  MoveL 2674 to (229.6, 36.16, 50.44) mm, rotated rx -180 ry 0 rz 180 deg; joints [-27.455, 46.759, -73.474, 30.185, 113.51, 13.063]
  Call Extruder(589.48218)
  MoveL 2675 to (229.82, 36.23, 50.44) mm, rotated rx -180 ry 0 rz 180 deg; joints [-27.424, 46.781, -73.473, 30.147, 113.498, 13.038]
  MoveL 2676 to (229.82, 36.23, 50.44) mm, rotated rx -180 ry 0 rz 180 deg; joints [-27.424, 46.781, -73.473, 30.147, 113.498, 13.038]
  Call Extruder(589.60868)
  MoveL 2677 to (230.04, 36.29, 50.44) mm, rotated rx -180 ry 0 rz 180 deg; joints [-27.392, 46.804, -73.473, 30.108, 113.485, 13.012]
  MoveL 2678 to (230.04, 36.29, 50.44) mm, rotated rx -180 ry 0 rz 180 deg; joints [-27.392, 46.804, -73.473, 30.108, 113.485, 13.012]
  Call Extruder(589.73571)
  MoveL 2679 to (230.26, 36.36, 50.44) mm, rotated rx 180 ry 0 rz 180 deg; joints [-27.361, 46.826, -73.473, 30.07, 113.473, 12.986]
  MoveL 2680 to (230.26, 36.36, 50.44) mm, rotated rx 180 ry 0 rz 180 deg; joints [-27.361, 46.826, -73.473, 30.07, 113.473, 12.986]
  Call Extruder(589.86325)
  MoveL 2681 to (230.48, 36.42, 50.44) mm, rotated rx -180 ry 0 rz 180 deg; joints [-27.33, 46.848, -73.472, 30.032, 113.46, 12.961]
  MoveL 2682 to (230.48, 36.42, 50.44) mm, rotated rx -180 ry 0 rz 180 deg; joints [-27.33, 46.848, -73.472, 30.032, 113.46, 12.961]
  Call Extruder(589.99132)
  MoveL 2683 to (230.7, 36.49, 50.44) mm, rotated rx 180 ry 0 rz 180 deg; joints [-27.299, 46.87, -73.472, 29.994, 113.448, 12.935]
  MoveL 2684 to (230.7, 36.49, 50.44) mm, rotated rx 180 ry 0 rz 180 deg; joints [-27.299, 46.87, -73.472, 29.994, 113.448, 12.935]
  Call Extruder(590.10322)
  MoveL 2685 to (230.88, 36.55, 50.44) mm, rotated rx -180 ry 0 rz 180 deg; joints [-27.276, 46.89, -73.472, 29.966, 113.436, 12.915]
  MoveL 2686 to (230.88, 36.55, 50.44) mm, rotated rx -180 ry 0 rz 180 deg; joints [-27.276, 46.89, -73.472, 29.966, 113.436, 12.915]
  Call Extruder(590.21556)
  MoveL 2687 to (231.07, 36.61, 50.44) mm, rotated rx -180 ry 0 rz 180 deg; joints [-27.253, 46.909, -73.471, 29.937, 113.424, 12.894]
  MoveL 2688 to (231.07, 36.61, 50.44) mm, rotated rx -180 ry 0 rz 180 deg; joints [-27.253, 46.909, -73.471, 29.937, 113.424, 12.894]
  Call Extruder(590.32835)
  MoveL 2689 to (231.26, 36.67, 50.44) mm, rotated rx -180 ry 0 rz -180 deg; joints [-27.231, 46.929, -73.471, 29.909, 113.412, 12.874]
  MoveL 2690 to (231.26, 36.67, 50.44) mm, rotated rx -180 ry 0 rz -180 deg; joints [-27.231, 46.929, -73.471, 29.909, 113.412, 12.874]
  Call Extruder(590.44158)
  MoveL 2691 to (231.45, 36.73, 50.44) mm, rotated rx -180 ry 0 rz 180 deg; joints [-27.208, 46.948, -73.47, 29.88, 113.399, 12.854]
  MoveL 2692 to (231.45, 36.73, 50.44) mm, rotated rx -180 ry 0 rz 180 deg; joints [-27.208, 46.948, -73.47, 29.88, 113.399, 12.854]
  Call Extruder(590.55526)
  MoveL 2693 to (231.64, 36.79, 50.44) mm, rotated rx 180 ry 0 rz 180 deg; joints [-27.185, 46.967, -73.47, 29.852, 113.387, 12.834]
  MoveL 2694 to (231.64, 36.79, 50.44) mm, rotated rx 180 ry 0 rz 180 deg; joints [-27.185, 46.967, -73.47, 29.852, 113.387, 12.834]
  Call Extruder(590.73722)
  MoveL 2695 to (231.93, 36.91, 50.44) mm, rotated rx -180 ry 0 rz 180 deg; joints [-27.167, 46.999, -73.469, 29.826, 113.364, 12.809]
  MoveL 2696 to (231.93, 36.91, 50.44) mm, rotated rx -180 ry 0 rz 180 deg; joints [-27.167, 46.999, -73.469, 29.826, 113.364, 12.809]
  Call Extruder(590.91994)
  MoveL 2697 to (232.22, 37.04, 50.44) mm, rotated rx -180 ry 0 rz 180 deg; joints [-27.149, 47.03, -73.469, 29.8, 113.34, 12.784]
  MoveL 2698 to (232.22, 37.04, 50.44) mm, rotated rx -180 ry 0 rz 180 deg; joints [-27.149, 47.03, -73.469, 29.8, 113.34, 12.784]
  Call Extruder(591.09035)
  MoveL 2699 to (232.49, 37.15, 50.44) mm, rotated rx -180 ry 0 rz 180 deg; joints [-27.133, 47.059, -73.468, 29.777, 113.318, 12.761]
  MoveL 2700 to (232.49, 37.15, 50.44) mm, rotated rx -180 ry 0 rz 180 deg; joints [-27.133, 47.059, -73.468, 29.777, 113.318, 12.761]
  Call Extruder(591.24835)
  MoveL 2701 to (232.74, 37.26, 50.44) mm, rotated rx -180 ry 0 rz 180 deg; joints [-27.121, 47.085, -73.467, 29.758, 113.297, 12.741]
  MoveL 2702 to (232.74, 37.26, 50.44) mm, rotated rx -180 ry 0 rz 180 deg; joints [-27.121, 47.085, -73.467, 29.758, 113.297, 12.741]
  Call Extruder(591.40695)
  MoveL 2703 to (232.99, 37.36, 50.44) mm, rotated rx -180 ry 0 rz -180 deg; joints [-27.108, 47.112, -73.467, 29.738, 113.276, 12.721]
  MoveL 2704 to (232.99, 37.36, 50.44) mm, rotated rx -180 ry 0 rz -180 deg; joints [-27.108, 47.112, -73.467, 29.738, 113.276, 12.721]
  Call Extruder(591.61312)
  MoveL 2705 to (233.29, 37.54, 50.44) mm, rotated rx 180 ry 0 rz -180 deg; joints [-27.12, 47.147, -73.466, 29.743, 113.242, 12.707]
  MoveL 2706 to (233.29, 37.54, 50.44) mm, rotated rx 180 ry 0 rz -180 deg; joints [-27.12, 47.147, -73.466, 29.743, 113.242, 12.707]
  Call Extruder(591.82006)
  MoveL 2707 to (233.6, 37.71, 50.44) mm, rotated rx 180 ry 0 rz -180 deg; joints [-27.132, 47.181, -73.465, 29.749, 113.209, 12.693]
  MoveL 2708 to (233.6, 37.71, 50.44) mm, rotated rx 180 ry 0 rz -180 deg; joints [-27.132, 47.181, -73.465, 29.749, 113.209, 12.693]
  Call Extruder(592.02779)
  MoveL 2709 to (233.9, 37.89, 50.44) mm, rotated rx -180 ry 0 rz 180 deg; joints [-27.144, 47.216, -73.464, 29.754, 113.175, 12.678]
  MoveL 2710 to (233.9, 37.89, 50.44) mm, rotated rx -180 ry 0 rz 180 deg; joints [-27.144, 47.216, -73.464, 29.754, 113.175, 12.678]
  Call Extruder(592.23629)
  MoveL 2711 to (234.21, 38.07, 50.44) mm, rotated rx 180 ry 0 rz -180 deg; joints [-27.156, 47.251, -73.462, 29.759, 113.141, 12.664]
  MoveL 2712 to (234.21, 38.07, 50.44) mm, rotated rx 180 ry 0 rz -180 deg; joints [-27.156, 47.251, -73.462, 29.759, 113.141, 12.664]
  Call Extruder(592.41583)
  MoveL 2713 to (234.45, 38.24, 50.44) mm, rotated rx 180 ry 0 rz 180 deg; joints [-27.187, 47.28, -73.461, 29.785, 113.108, 12.661]
  MoveL 2714 to (234.45, 38.24, 50.44) mm, rotated rx 180 ry 0 rz 180 deg; joints [-27.187, 47.28, -73.461, 29.785, 113.108, 12.661]
  Call Extruder(592.74925)
  MoveL 2715 to (234.9, 38.57, 50.44) mm, rotated rx -180 ry 0 rz 180 deg; joints [-27.245, 47.334, -73.46, 29.835, 113.047, 12.655]
  MoveL 2716 to (234.9, 38.57, 50.44) mm, rotated rx -180 ry 0 rz 180 deg; joints [-27.245, 47.334, -73.46, 29.835, 113.047, 12.655]
  Call Extruder(593.08385)
  MoveL 2717 to (235.35, 38.9, 50.44) mm, rotated rx 180 ry 0 rz 180 deg; joints [-27.302, 47.388, -73.458, 29.884, 112.986, 12.648]
  Call Extruder(593.91180)
  MoveL 2718 to (236.39, 39.81, 50.44) mm, rotated rx -180 ry 0 rz 180 deg; joints [-27.525, 47.52, -73.452, 30.091, 112.819, 12.665]
  Call Extruder(594.73974)
  MoveL 2719 to (237.3, 40.85, 50.44) mm, rotated rx -180 ry 0 rz 180 deg; joints [-27.851, 47.646, -73.447, 30.408, 112.633, 12.727]
  Call Extruder(594.90704)
  MoveL 2720 to (237.47, 41.07, 50.44) mm, rotated rx -180 ry 0 rz 180 deg; joints [-27.932, 47.67, -73.445, 30.488, 112.593, 12.745]
  MoveL 2721 to (237.47, 41.07, 50.44) mm, rotated rx -180 ry 0 rz 180 deg; joints [-27.932, 47.67, -73.445, 30.488, 112.593, 12.745]
  Call Extruder(595.24045)
  MoveL 2722 to (237.8, 41.52, 50.44) mm, rotated rx 180 ry 0 rz -180 deg; joints [-28.091, 47.719, -73.443, 30.645, 112.514, 12.782]
  MoveL 2723 to (237.8, 41.52, 50.44) mm, rotated rx 180 ry 0 rz -180 deg; joints [-28.091, 47.719, -73.443, 30.645, 112.514, 12.782]
  Call Extruder(595.57268)
  MoveL 2724 to (238.12, 41.98, 50.44) mm, rotated rx -180 ry 0 rz 180 deg; joints [-28.249, 47.768, -73.44, 30.801, 112.434, 12.817]
  MoveL 2725 to (238.12, 41.98, 50.44) mm, rotated rx -180 ry 0 rz 180 deg; joints [-28.249, 47.768, -73.44, 30.801, 112.434, 12.817]
  Call Extruder(595.69039)
  MoveL 2726 to (238.22, 42.15, 50.44) mm, rotated rx -180 ry 0 rz 180 deg; joints [-28.315, 47.784, -73.439, 30.867, 112.405, 12.834]
  MoveL 2727 to (238.22, 42.15, 50.44) mm, rotated rx -180 ry 0 rz 180 deg; joints [-28.315, 47.784, -73.439, 30.867, 112.405, 12.834]
  Call Extruder(595.89811)
  MoveL 2728 to (238.4, 42.45, 50.44) mm, rotated rx 180 ry 0 rz 180 deg; joints [-28.434, 47.814, -73.438, 30.986, 112.352, 12.864]
  MoveL 2729 to (238.4, 42.45, 50.44) mm, rotated rx 180 ry 0 rz 180 deg; joints [-28.434, 47.814, -73.438, 30.986, 112.352, 12.864]
  Call Extruder(596.10507)
  MoveL 2730 to (238.57, 42.75, 50.44) mm, rotated rx 180 ry 0 rz 180 deg; joints [-28.552, 47.843, -73.436, 31.103, 112.3, 12.895]
  MoveL 2731 to (238.57, 42.75, 50.44) mm, rotated rx 180 ry 0 rz 180 deg; joints [-28.552, 47.843, -73.436, 31.103, 112.3, 12.895]
  Call Extruder(596.31124)
  MoveL 2732 to (238.75, 43.06, 50.44) mm, rotated rx -180 ry 0 rz 180 deg; joints [-28.669, 47.872, -73.435, 31.22, 112.247, 12.924]
  MoveL 2733 to (238.75, 43.06, 50.44) mm, rotated rx -180 ry 0 rz 180 deg; joints [-28.669, 47.872, -73.435, 31.22, 112.247, 12.924]
  Call Extruder(596.49292)
  MoveL 2734 to (238.89, 43.34, 50.44) mm, rotated rx -180 ry 0 rz 180 deg; joints [-28.78, 47.897, -73.433, 31.332, 112.2, 12.954]
  MoveL 2735 to (238.89, 43.34, 50.44) mm, rotated rx -180 ry 0 rz 180 deg; joints [-28.78, 47.897, -73.433, 31.332, 112.2, 12.954]
  Call Extruder(596.65093)
  MoveL 2736 to (239, 43.58, 50.44) mm, rotated rx 180 ry 0 rz 180 deg; joints [-28.886, 47.917, -73.432, 31.439, 112.157, 12.983]
  MoveL 2737 to (239, 43.58, 50.44) mm, rotated rx 180 ry 0 rz 180 deg; joints [-28.886, 47.917, -73.432, 31.439, 112.157, 12.983]
  Call Extruder(596.80833)
  MoveL 2738 to (239.11, 43.83, 50.44) mm, rotated rx -180 ry 0 rz 180 deg; joints [-28.991, 47.938, -73.431, 31.545, 112.115, 13.013]
  MoveL 2739 to (239.11, 43.83, 50.44) mm, rotated rx -180 ry 0 rz 180 deg; joints [-28.991, 47.938, -73.431, 31.545, 112.115, 13.013]
  Call Extruder(596.98254)
  MoveL 2740 to (239.22, 44.11, 50.44) mm, rotated rx -180 ry 0 rz 180 deg; joints [-29.11, 47.961, -73.429, 31.664, 112.067, 13.046]
  MoveL 2741 to (239.22, 44.11, 50.44) mm, rotated rx -180 ry 0 rz 180 deg; joints [-29.11, 47.961, -73.429, 31.664, 112.067, 13.046]
  Call Extruder(597.15607)
  MoveL 2742 to (239.33, 44.39, 50.44) mm, rotated rx -180 ry 0 rz 180 deg; joints [-29.228, 47.984, -73.428, 31.783, 112.02, 13.079]
  MoveL 2743 to (239.33, 44.39, 50.44) mm, rotated rx -180 ry 0 rz 180 deg; joints [-29.228, 47.984, -73.428, 31.783, 112.02, 13.079]
  Call Extruder(597.26356)
  MoveL 2744 to (239.41, 44.56, 50.44) mm, rotated rx -180 ry 0 rz 180 deg; joints [-29.301, 47.998, -73.427, 31.857, 111.991, 13.099]
  MoveL 2745 to (239.41, 44.56, 50.44) mm, rotated rx -180 ry 0 rz 180 deg; joints [-29.301, 47.998, -73.427, 31.857, 111.991, 13.099]
  Call Extruder(597.37703)
  MoveL 2746 to (239.47, 44.75, 50.44) mm, rotated rx -180 ry 0 rz -180 deg; joints [-29.385, 48.012, -73.426, 31.942, 111.959, 13.123]
  MoveL 2747 to (239.47, 44.75, 50.44) mm, rotated rx -180 ry 0 rz -180 deg; joints [-29.385, 48.012, -73.426, 31.942, 111.959, 13.123]
  Call Extruder(597.49005)
  MoveL 2748 to (239.53, 44.94, 50.44) mm, rotated rx -180 ry 0 rz 180 deg; joints [-29.47, 48.026, -73.425, 32.028, 111.927, 13.148]
  MoveL 2749 to (239.53, 44.94, 50.44) mm, rotated rx -180 ry 0 rz 180 deg; joints [-29.47, 48.026, -73.425, 32.028, 111.927, 13.148]
  Call Extruder(597.60263)
  MoveL 2750 to (239.59, 45.13, 50.44) mm, rotated rx 180 ry 0 rz -180 deg; joints [-29.553, 48.041, -73.424, 32.112, 111.895, 13.172]
  MoveL 2751 to (239.59, 45.13, 50.44) mm, rotated rx 180 ry 0 rz -180 deg; joints [-29.553, 48.041, -73.424, 32.112, 111.895, 13.172]
  Call Extruder(597.71477)
  MoveL 2752 to (239.65, 45.32, 50.44) mm, rotated rx 180 ry 0 rz 180 deg; joints [-29.637, 48.055, -73.423, 32.197, 111.863, 13.196]
  MoveL 2753 to (239.65, 45.32, 50.44) mm, rotated rx 180 ry 0 rz 180 deg; joints [-29.637, 48.055, -73.423, 32.197, 111.863, 13.196]
  Call Extruder(597.82645)
  MoveL 2754 to (239.71, 45.5, 50.44) mm, rotated rx -180 ry 0 rz 180 deg; joints [-29.72, 48.069, -73.422, 32.281, 111.831, 13.22]
  MoveL 2755 to (239.71, 45.5, 50.44) mm, rotated rx -180 ry 0 rz 180 deg; joints [-29.72, 48.069, -73.422, 32.281, 111.831, 13.22]
  Call Extruder(597.95753)
  MoveL 2756 to (239.78, 45.73, 50.44) mm, rotated rx 180 ry 0 rz 180 deg; joints [-29.821, 48.085, -73.421, 32.382, 111.794, 13.249]
  MoveL 2757 to (239.78, 45.73, 50.44) mm, rotated rx 180 ry 0 rz 180 deg; joints [-29.821, 48.085, -73.421, 32.382, 111.794, 13.249]
  Call Extruder(598.08804)
  MoveL 2758 to (239.85, 45.95, 50.44) mm, rotated rx 180 ry 0 rz 180 deg; joints [-29.921, 48.102, -73.42, 32.483, 111.756, 13.278]
  MoveL 2759 to (239.85, 45.95, 50.44) mm, rotated rx 180 ry 0 rz 180 deg; joints [-29.921, 48.102, -73.42, 32.483, 111.756, 13.278]
  Call Extruder(598.21798)
  MoveL 2760 to (239.92, 46.18, 50.44) mm, rotated rx -180 ry 0 rz 180 deg; joints [-30.02, 48.118, -73.419, 32.583, 111.718, 13.306]
  MoveL 2761 to (239.92, 46.18, 50.44) mm, rotated rx -180 ry 0 rz 180 deg; joints [-30.02, 48.118, -73.419, 32.583, 111.718, 13.306]
  Call Extruder(598.34736)
  MoveL 2762 to (239.98, 46.4, 50.44) mm, rotated rx 180 ry 0 rz -180 deg; joints [-30.119, 48.135, -73.418, 32.683, 111.681, 13.334]
  MoveL 2763 to (239.98, 46.4, 50.44) mm, rotated rx 180 ry 0 rz -180 deg; joints [-30.119, 48.135, -73.418, 32.683, 111.681, 13.334]
  Call Extruder(598.46931)
  MoveL 2764 to (240.04, 46.61, 50.44) mm, rotated rx -180 ry 0 rz 180 deg; joints [-30.216, 48.15, -73.417, 32.781, 111.645, 13.362]
  MoveL 2765 to (240.04, 46.61, 50.44) mm, rotated rx -180 ry 0 rz 180 deg; joints [-30.216, 48.15, -73.417, 32.781, 111.645, 13.362]
  Call Extruder(598.58414)
  MoveL 2766 to (240.08, 46.82, 50.44) mm, rotated rx -180 ry 0 rz 180 deg; joints [-30.311, 48.163, -73.416, 32.878, 111.61, 13.391]
  MoveL 2767 to (240.08, 46.82, 50.44) mm, rotated rx -180 ry 0 rz 180 deg; joints [-30.311, 48.163, -73.416, 32.878, 111.61, 13.391]
  Call Extruder(598.69851)
  MoveL 2768 to (240.13, 47.02, 50.44) mm, rotated rx -180 ry 0 rz 180 deg; joints [-30.406, 48.177, -73.415, 32.974, 111.576, 13.418]
  MoveL 2769 to (240.13, 47.02, 50.44) mm, rotated rx -180 ry 0 rz 180 deg; joints [-30.406, 48.177, -73.415, 32.974, 111.576, 13.418]
  Call Extruder(598.81243)
  MoveL 2770 to (240.17, 47.23, 50.44) mm, rotated rx -180 ry 0 rz 180 deg; joints [-30.5, 48.191, -73.414, 33.069, 111.542, 13.446]
  MoveL 2771 to (240.17, 47.23, 50.44) mm, rotated rx -180 ry 0 rz 180 deg; joints [-30.5, 48.191, -73.414, 33.069, 111.542, 13.446]
  Call Extruder(598.92591)
  MoveL 2772 to (240.22, 47.43, 50.44) mm, rotated rx -180 ry 0 rz 180 deg; joints [-30.595, 48.204, -73.413, 33.165, 111.508, 13.474]
  MoveL 2773 to (240.22, 47.43, 50.44) mm, rotated rx -180 ry 0 rz 180 deg; joints [-30.595, 48.204, -73.413, 33.165, 111.508, 13.474]
  Call Extruder(599.06319)
  MoveL 2774 to (240.27, 47.68, 50.44) mm, rotated rx -180 ry 0 rz 180 deg; joints [-30.711, 48.221, -73.412, 33.283, 111.466, 13.508]
  MoveL 2775 to (240.27, 47.68, 50.44) mm, rotated rx -180 ry 0 rz 180 deg; joints [-30.711, 48.221, -73.412, 33.283, 111.466, 13.508]
  Call Extruder(599.19986)
  MoveL 2776 to (240.32, 47.93, 50.44) mm, rotated rx -180 ry 0 rz 180 deg; joints [-30.827, 48.237, -73.411, 33.4, 111.424, 13.542]
  MoveL 2777 to (240.32, 47.93, 50.44) mm, rotated rx -180 ry 0 rz 180 deg; joints [-30.827, 48.237, -73.411, 33.4, 111.424, 13.542]
  Call Extruder(599.33592)
  MoveL 2778 to (240.37, 48.18, 50.44) mm, rotated rx -180 ry 0 rz 180 deg; joints [-30.942, 48.253, -73.409, 33.516, 111.383, 13.575]
  MoveL 2779 to (240.37, 48.18, 50.44) mm, rotated rx -180 ry 0 rz 180 deg; joints [-30.942, 48.253, -73.409, 33.516, 111.383, 13.575]
  Call Extruder(599.47137)
  MoveL 2780 to (240.42, 48.43, 50.44) mm, rotated rx -180 ry 0 rz 180 deg; joints [-31.057, 48.27, -73.408, 33.632, 111.341, 13.608]
  MoveL 2781 to (240.42, 48.43, 50.44) mm, rotated rx -180 ry 0 rz 180 deg; joints [-31.057, 48.27, -73.408, 33.632, 111.341, 13.608]
  Call Extruder(599.60622)
  MoveL 2782 to (240.47, 48.68, 50.44) mm, rotated rx 180 ry 0 rz 180 deg; joints [-31.171, 48.286, -73.407, 33.748, 111.299, 13.641]
  MoveL 2783 to (240.47, 48.68, 50.44) mm, rotated rx 180 ry 0 rz 180 deg; joints [-31.171, 48.286, -73.407, 33.748, 111.299, 13.641]
  Call Extruder(599.74045)
  MoveL 2784 to (240.52, 48.92, 50.44) mm, rotated rx -180 ry 0 rz 180 deg; joints [-31.285, 48.303, -73.406, 33.863, 111.258, 13.674]
  MoveL 2785 to (240.52, 48.92, 50.44) mm, rotated rx -180 ry 0 rz 180 deg; joints [-31.285, 48.303, -73.406, 33.863, 111.258, 13.674]
  Call Extruder(599.87407)
  MoveL 2786 to (240.57, 49.17, 50.44) mm, rotated rx -180 ry 0 rz 180 deg; joints [-31.398, 48.319, -73.405, 33.977, 111.216, 13.706]
  MoveL 2787 to (240.57, 49.17, 50.44) mm, rotated rx -180 ry 0 rz 180 deg; joints [-31.398, 48.319, -73.405, 33.977, 111.216, 13.706]
  Call Extruder(600.03618)
  MoveL 2788 to (240.61, 49.48, 50.44) mm, rotated rx 180 ry 0 rz 180 deg; joints [-31.541, 48.339, -73.403, 34.121, 111.165, 13.747]
  MoveL 2789 to (240.61, 49.48, 50.44) mm, rotated rx 180 ry 0 rz 180 deg; joints [-31.541, 48.339, -73.403, 34.121, 111.165, 13.747]
  Call Extruder(600.19756)
  MoveL 2790 to (240.66, 49.79, 50.44) mm, rotated rx -180 ry 0 rz 180 deg; joints [-31.684, 48.358, -73.402, 34.265, 111.114, 13.788]
  MoveL 2791 to (240.66, 49.79, 50.44) mm, rotated rx -180 ry 0 rz 180 deg; joints [-31.684, 48.358, -73.402, 34.265, 111.114, 13.788]
  Call Extruder(600.35821)
  MoveL 2792 to (240.71, 50.09, 50.44) mm, rotated rx -180 ry 0 rz 180 deg; joints [-31.825, 48.377, -73.4, 34.408, 111.063, 13.829]
  MoveL 2793 to (240.71, 50.09, 50.44) mm, rotated rx -180 ry 0 rz 180 deg; joints [-31.825, 48.377, -73.4, 34.408, 111.063, 13.829]
  Call Extruder(600.51814)
  MoveL 2794 to (240.76, 50.4, 50.44) mm, rotated rx -180 ry 0 rz 180 deg; joints [-31.966, 48.397, -73.398, 34.55, 111.012, 13.868]
  MoveL 2795 to (240.76, 50.4, 50.44) mm, rotated rx -180 ry 0 rz 180 deg; joints [-31.966, 48.397, -73.398, 34.55, 111.012, 13.868]
  Call Extruder(600.67734)
  MoveL 2796 to (240.81, 50.7, 50.44) mm, rotated rx -180 ry 0 rz 180 deg; joints [-32.106, 48.416, -73.397, 34.691, 110.961, 13.908]
  MoveL 2797 to (240.81, 50.7, 50.44) mm, rotated rx -180 ry 0 rz 180 deg; joints [-32.106, 48.416, -73.397, 34.691, 110.961, 13.908]
  Call Extruder(600.83580)
  MoveL 2798 to (240.86, 51.01, 50.44) mm, rotated rx 180 ry 0 rz 180 deg; joints [-32.246, 48.436, -73.395, 34.832, 110.91, 13.947]
  MoveL 2799 to (240.86, 51.01, 50.44) mm, rotated rx 180 ry 0 rz 180 deg; joints [-32.246, 48.436, -73.395, 34.832, 110.91, 13.947]
  Call Extruder(601.03468)
  MoveL 2800 to (240.9, 51.4, 50.44) mm, rotated rx -180 ry 0 rz 180 deg; joints [-32.427, 48.459, -73.393, 35.015, 110.845, 13.998]
  MoveL 2801 to (240.9, 51.4, 50.44) mm, rotated rx -180 ry 0 rz 180 deg; joints [-32.427, 48.459, -73.393, 35.015, 110.845, 13.998]
  Call Extruder(601.23269)
  MoveL 2802 to (240.95, 51.78, 50.44) mm, rotated rx -180 ry 0 rz 180 deg; joints [-32.608, 48.483, -73.391, 35.196, 110.78, 14.049]
  MoveL 2803 to (240.95, 51.78, 50.44) mm, rotated rx -180 ry 0 rz 180 deg; joints [-32.608, 48.483, -73.391, 35.196, 110.78, 14.049]
  Call Extruder(601.42983)
  MoveL 2804 to (240.99, 52.17, 50.44) mm, rotated rx -180 ry 0 rz 180 deg; joints [-32.787, 48.507, -73.389, 35.377, 110.716, 14.099]
  MoveL 2805 to (240.99, 52.17, 50.44) mm, rotated rx -180 ry 0 rz 180 deg; joints [-32.787, 48.507, -73.389, 35.377, 110.716, 14.099]
  Call Extruder(601.62610)
  MoveL 2806 to (241.04, 52.56, 50.44) mm, rotated rx -180 ry 0 rz -180 deg; joints [-32.966, 48.53, -73.387, 35.556, 110.651, 14.149]
  MoveL 2807 to (241.04, 52.56, 50.44) mm, rotated rx -180 ry 0 rz -180 deg; joints [-32.966, 48.53, -73.387, 35.556, 110.651, 14.149]
  Call Extruder(601.87181)
  MoveL 2808 to (241.09, 53.05, 50.44) mm, rotated rx 180 ry 0 rz 180 deg; joints [-33.193, 48.56, -73.385, 35.785, 110.57, 14.212]
  MoveL 2809 to (241.09, 53.05, 50.44) mm, rotated rx 180 ry 0 rz 180 deg; joints [-33.193, 48.56, -73.385, 35.785, 110.57, 14.212]
  Call Extruder(602.16658)
  MoveL 2810 to (241.13, 53.64, 50.44) mm, rotated rx 180 ry 0 rz 180 deg; joints [-33.469, 48.594, -73.382, 36.062, 110.471, 14.288]
  MoveL 2811 to (241.13, 53.64, 50.44) mm, rotated rx 180 ry 0 rz 180 deg; joints [-33.469, 48.594, -73.382, 36.062, 110.471, 14.288]
  Call Extruder(602.46002)
  MoveL 2812 to (241.18, 54.23, 50.44) mm, rotated rx -180 ry 0 rz 180 deg; joints [-33.742, 48.629, -73.379, 36.336, 110.373, 14.363]
  MoveL 2813 to (241.18, 54.23, 50.44) mm, rotated rx -180 ry 0 rz 180 deg; joints [-33.742, 48.629, -73.379, 36.336, 110.373, 14.363]
  Call Extruder(602.89337)
  MoveL 2814 to (241.23, 55.1, 50.44) mm, rotated rx -180 ry 0 rz 180 deg; joints [-34.152, 48.679, -73.374, 36.748, 110.227, 14.475]
  MoveL 2815 to (241.23, 55.1, 50.44) mm, rotated rx -180 ry 0 rz 180 deg; joints [-34.152, 48.679, -73.374, 36.748, 110.227, 14.475]
  Call Extruder(603.46554)
  MoveL 2816 to (241.27, 56.26, 50.44) mm, rotated rx -180 ry 0 rz 180 deg; joints [-34.696, 48.745, -73.368, 37.292, 110.033, 14.621]
  MoveL 2817 to (241.27, 56.26, 50.44) mm, rotated rx -180 ry 0 rz 180 deg; joints [-34.696, 48.745, -73.368, 37.292, 110.033, 14.621]
  Call Extruder(603.89324)
  MoveL 2818 to (241.29, 57.14, 50.44) mm, rotated rx 180 ry 0 rz 180 deg; joints [-35.104, 48.794, -73.363, 37.7, 109.887, 14.73]
  Call Extruder(645.88687)
  MoveL 2819 to (241.29, 142.86, 50.44) mm, rotated rx 180 ry 0 rz 180 deg; joints [-60.361, 54.458, -71.96, 61.513, 98.553, 15.326]
  MoveL 2820 to (241.29, 142.86, 50.44) mm, rotated rx 180 ry 0 rz 180 deg; joints [-60.361, 54.458, -71.96, 61.513, 98.553, 15.326]
  Call Extruder(646.60231)
  MoveL 2821 to (241.25, 144.32, 50.44) mm, rotated rx 180 ry 0 rz 180 deg; joints [-60.621, 54.556, -71.917, 61.749, 98.417, 15.239]
  MoveL 2822 to (241.25, 144.32, 50.44) mm, rotated rx 180 ry 0 rz 180 deg; joints [-60.621, 54.556, -71.917, 61.749, 98.417, 15.239]
  Call Extruder(647.17705)
  MoveL 2823 to (241.2, 145.48, 50.44) mm, rotated rx -180 ry 0 rz 180 deg; joints [-60.831, 54.634, -71.883, 61.939, 98.309, 15.169]
  MoveL 2824 to (241.2, 145.48, 50.44) mm, rotated rx -180 ry 0 rz 180 deg; joints [-60.831, 54.634, -71.883, 61.939, 98.309, 15.169]
  Call Extruder(647.47049)
  MoveL 2825 to (241.16, 146.07, 50.44) mm, rotated rx -180 ry 0 rz 180 deg; joints [-60.944, 54.673, -71.865, 62.042, 98.254, 15.135]
  MoveL 2826 to (241.16, 146.07, 50.44) mm, rotated rx -180 ry 0 rz 180 deg; joints [-60.944, 54.673, -71.865, 62.042, 98.254, 15.135]
  Call Extruder(647.76527)
  MoveL 2827 to (241.11, 146.66, 50.44) mm, rotated rx -180 ry 0 rz 180 deg; joints [-61.055, 54.711, -71.848, 62.144, 98.198, 15.1]
  MoveL 2828 to (241.11, 146.66, 50.44) mm, rotated rx -180 ry 0 rz 180 deg; joints [-61.055, 54.711, -71.848, 62.144, 98.198, 15.1]
  Call Extruder(648.06138)
  MoveL 2829 to (241.06, 147.25, 50.44) mm, rotated rx -180 ry 0 rz -180 deg; joints [-61.167, 54.75, -71.831, 62.245, 98.143, 15.066]
  MoveL 2830 to (241.06, 147.25, 50.44) mm, rotated rx -180 ry 0 rz -180 deg; joints [-61.167, 54.75, -71.831, 62.245, 98.143, 15.066]
  Call Extruder(648.25765)
  MoveL 2831 to (241.02, 147.63, 50.44) mm, rotated rx -180 ry 0 rz 180 deg; joints [-61.244, 54.775, -71.819, 62.316, 98.107, 15.044]
  MoveL 2832 to (241.02, 147.63, 50.44) mm, rotated rx -180 ry 0 rz 180 deg; joints [-61.244, 54.775, -71.819, 62.316, 98.107, 15.044]
  Call Extruder(648.45479)
  MoveL 2833 to (240.97, 148.02, 50.44) mm, rotated rx 180 ry 0 rz 180 deg; joints [-61.321, 54.799, -71.808, 62.386, 98.07, 15.023]
  MoveL 2834 to (240.97, 148.02, 50.44) mm, rotated rx 180 ry 0 rz 180 deg; joints [-61.321, 54.799, -71.808, 62.386, 98.07, 15.023]
  Call Extruder(648.65280)
  MoveL 2835 to (240.93, 148.41, 50.44) mm, rotated rx 180 ry 0 rz 180 deg; joints [-61.397, 54.824, -71.797, 62.457, 98.033, 15.001]
  MoveL 2836 to (240.93, 148.41, 50.44) mm, rotated rx 180 ry 0 rz 180 deg; joints [-61.397, 54.824, -71.797, 62.457, 98.033, 15.001]
  Call Extruder(648.85167)
  MoveL 2837 to (240.88, 148.8, 50.44) mm, rotated rx -180 ry 0 rz 180 deg; joints [-61.474, 54.849, -71.785, 62.527, 97.997, 14.979]
  MoveL 2838 to (240.88, 148.8, 50.44) mm, rotated rx -180 ry 0 rz 180 deg; joints [-61.474, 54.849, -71.785, 62.527, 97.997, 14.979]
  Call Extruder(649.03075)
  MoveL 2839 to (240.83, 149.14, 50.44) mm, rotated rx -180 ry 0 rz 180 deg; joints [-61.544, 54.871, -71.775, 62.591, 97.964, 14.96]
  MoveL 2840 to (240.83, 149.14, 50.44) mm, rotated rx -180 ry 0 rz 180 deg; joints [-61.544, 54.871, -71.775, 62.591, 97.964, 14.96]
  Call Extruder(649.18995)
  MoveL 2841 to (240.78, 149.45, 50.44) mm, rotated rx -180 ry 0 rz 180 deg; joints [-61.607, 54.89, -71.766, 62.649, 97.935, 14.943]
  MoveL 2842 to (240.78, 149.45, 50.44) mm, rotated rx -180 ry 0 rz 180 deg; joints [-61.607, 54.89, -71.766, 62.649, 97.935, 14.943]
  Call Extruder(649.34987)
  MoveL 2843 to (240.74, 149.76, 50.44) mm, rotated rx -180 ry 0 rz 180 deg; joints [-61.67, 54.909, -71.757, 62.708, 97.906, 14.927]
  MoveL 2844 to (240.74, 149.76, 50.44) mm, rotated rx -180 ry 0 rz 180 deg; joints [-61.67, 54.909, -71.757, 62.708, 97.906, 14.927]
  Call Extruder(649.51052)
  MoveL 2845 to (240.69, 150.06, 50.44) mm, rotated rx -180 ry 0 rz 180 deg; joints [-61.734, 54.928, -71.749, 62.766, 97.877, 14.91]
  MoveL 2846 to (240.69, 150.06, 50.44) mm, rotated rx -180 ry 0 rz 180 deg; joints [-61.734, 54.928, -71.749, 62.766, 97.877, 14.91]
  Call Extruder(649.67190)
  MoveL 2847 to (240.64, 150.37, 50.44) mm, rotated rx -180 ry 0 rz -180 deg; joints [-61.796, 54.947, -71.74, 62.824, 97.848, 14.893]
  MoveL 2848 to (240.64, 150.37, 50.44) mm, rotated rx -180 ry 0 rz -180 deg; joints [-61.796, 54.947, -71.74, 62.824, 97.848, 14.893]
  Call Extruder(649.83401)
  MoveL 2849 to (240.59, 150.67, 50.44) mm, rotated rx -180 ry 0 rz 180 deg; joints [-61.859, 54.966, -71.731, 62.882, 97.819, 14.876]
  MoveL 2850 to (240.59, 150.67, 50.44) mm, rotated rx -180 ry 0 rz 180 deg; joints [-61.859, 54.966, -71.731, 62.882, 97.819, 14.876]
  Call Extruder(649.98221)
  MoveL 2851 to (240.54, 150.95, 50.44) mm, rotated rx 180 ry 0 rz 180 deg; joints [-61.918, 54.983, -71.723, 62.936, 97.792, 14.862]
  MoveL 2852 to (240.54, 150.95, 50.44) mm, rotated rx 180 ry 0 rz 180 deg; joints [-61.918, 54.983, -71.723, 62.936, 97.792, 14.862]
  Call Extruder(650.11644)
  MoveL 2853 to (240.49, 151.2, 50.44) mm, rotated rx -180 ry 0 rz 180 deg; joints [-61.971, 54.998, -71.715, 62.985, 97.768, 14.848]
  MoveL 2854 to (240.49, 151.2, 50.44) mm, rotated rx -180 ry 0 rz 180 deg; joints [-61.971, 54.998, -71.715, 62.985, 97.768, 14.848]
  Call Extruder(650.25129)
  MoveL 2855 to (240.44, 151.45, 50.44) mm, rotated rx -180 ry 0 rz 180 deg; joints [-62.025, 55.013, -71.708, 63.035, 97.745, 14.836]
  MoveL 2856 to (240.44, 151.45, 50.44) mm, rotated rx -180 ry 0 rz 180 deg; joints [-62.025, 55.013, -71.708, 63.035, 97.745, 14.836]
  Call Extruder(650.38674)
  MoveL 2857 to (240.39, 151.7, 50.44) mm, rotated rx 180 ry 0 rz 180 deg; joints [-62.079, 55.028, -71.701, 63.084, 97.721, 14.822]
  MoveL 2858 to (240.39, 151.7, 50.44) mm, rotated rx 180 ry 0 rz 180 deg; joints [-62.079, 55.028, -71.701, 63.084, 97.721, 14.822]
  Call Extruder(650.52280)
  MoveL 2859 to (240.34, 151.95, 50.44) mm, rotated rx -180 ry 0 rz -180 deg; joints [-62.132, 55.044, -71.694, 63.134, 97.697, 14.809]
  MoveL 2860 to (240.34, 151.95, 50.44) mm, rotated rx -180 ry 0 rz -180 deg; joints [-62.132, 55.044, -71.694, 63.134, 97.697, 14.809]
  Call Extruder(650.65947)
  MoveL 2861 to (240.29, 152.2, 50.44) mm, rotated rx -180 ry 0 rz -180 deg; joints [-62.186, 55.059, -71.686, 63.183, 97.673, 14.796]
  MoveL 2862 to (240.29, 152.2, 50.44) mm, rotated rx -180 ry 0 rz -180 deg; joints [-62.186, 55.059, -71.686, 63.183, 97.673, 14.796]
  Call Extruder(650.79675)
  MoveL 2863 to (240.24, 152.44, 50.44) mm, rotated rx -180 ry 0 rz 180 deg; joints [-62.239, 55.074, -71.679, 63.233, 97.649, 14.783]
  MoveL 2864 to (240.24, 152.44, 50.44) mm, rotated rx -180 ry 0 rz 180 deg; joints [-62.239, 55.074, -71.679, 63.233, 97.649, 14.783]
  Call Extruder(650.92242)
  MoveL 2865 to (240.2, 152.67, 50.44) mm, rotated rx -180 ry 0 rz 180 deg; joints [-62.288, 55.088, -71.673, 63.278, 97.628, 14.771]
  MoveL 2866 to (240.2, 152.67, 50.44) mm, rotated rx -180 ry 0 rz 180 deg; joints [-62.288, 55.088, -71.673, 63.278, 97.628, 14.771]
  Call Extruder(651.03634)
  MoveL 2867 to (240.15, 152.88, 50.44) mm, rotated rx -180 ry 0 rz 180 deg; joints [-62.333, 55.1, -71.667, 63.319, 97.608, 14.76]
  MoveL 2868 to (240.15, 152.88, 50.44) mm, rotated rx -180 ry 0 rz 180 deg; joints [-62.333, 55.1, -71.667, 63.319, 97.608, 14.76]
  Call Extruder(651.15072)
  MoveL 2869 to (240.11, 153.08, 50.44) mm, rotated rx -180 ry 0 rz 180 deg; joints [-62.377, 55.112, -71.661, 63.36, 97.589, 14.749]
  MoveL 2870 to (240.11, 153.08, 50.44) mm, rotated rx -180 ry 0 rz 180 deg; joints [-62.377, 55.112, -71.661, 63.36, 97.589, 14.749]
  Call Extruder(651.26555)
  MoveL 2871 to (240.06, 153.28, 50.44) mm, rotated rx -180 ry 0 rz 180 deg; joints [-62.421, 55.124, -71.655, 63.402, 97.569, 14.739]
  MoveL 2872 to (240.06, 153.28, 50.44) mm, rotated rx -180 ry 0 rz 180 deg; joints [-62.421, 55.124, -71.655, 63.402, 97.569, 14.739]
  Call Extruder(651.38083)
  MoveL 2873 to (240.02, 153.49, 50.44) mm, rotated rx -180 ry 0 rz 180 deg; joints [-62.466, 55.137, -71.649, 63.443, 97.55, 14.728]
  MoveL 2874 to (240.02, 153.49, 50.44) mm, rotated rx -180 ry 0 rz 180 deg; joints [-62.466, 55.137, -71.649, 63.443, 97.55, 14.728]
  Call Extruder(651.51021)
  MoveL 2875 to (239.95, 153.71, 50.44) mm, rotated rx 180 ry 0 rz 180 deg; joints [-62.52, 55.15, -71.642, 63.493, 97.527, 14.718]
  MoveL 2876 to (239.95, 153.71, 50.44) mm, rotated rx 180 ry 0 rz 180 deg; joints [-62.52, 55.15, -71.642, 63.493, 97.527, 14.718]
  Call Extruder(651.64015)
  MoveL 2877 to (239.88, 153.94, 50.44) mm, rotated rx -180 ry 0 rz -180 deg; joints [-62.574, 55.162, -71.636, 63.544, 97.505, 14.707]
  MoveL 2878 to (239.88, 153.94, 50.44) mm, rotated rx -180 ry 0 rz -180 deg; joints [-62.574, 55.162, -71.636, 63.544, 97.505, 14.707]
  Call Extruder(651.77066)
  MoveL 2879 to (239.81, 154.16, 50.44) mm, rotated rx -180 ry 0 rz 180 deg; joints [-62.627, 55.175, -71.63, 63.594, 97.483, 14.697]
  MoveL 2880 to (239.81, 154.16, 50.44) mm, rotated rx -180 ry 0 rz 180 deg; joints [-62.627, 55.175, -71.63, 63.594, 97.483, 14.697]
  Call Extruder(651.90174)
  MoveL 2881 to (239.75, 154.38, 50.44) mm, rotated rx -180 ry 0 rz 180 deg; joints [-62.681, 55.188, -71.624, 63.644, 97.461, 14.686]
  MoveL 2882 to (239.75, 154.38, 50.44) mm, rotated rx -180 ry 0 rz 180 deg; joints [-62.681, 55.188, -71.624, 63.644, 97.461, 14.686]
  Call Extruder(652.02338)
  MoveL 2883 to (239.68, 154.59, 50.44) mm, rotated rx 180 ry 0 rz 180 deg; joints [-62.731, 55.2, -71.618, 63.691, 97.441, 14.677]
  MoveL 2884 to (239.68, 154.59, 50.44) mm, rotated rx 180 ry 0 rz 180 deg; joints [-62.731, 55.2, -71.618, 63.691, 97.441, 14.677]
  Call Extruder(652.13550)
  MoveL 2885 to (239.62, 154.78, 50.44) mm, rotated rx 180 ry 0 rz 180 deg; joints [-62.778, 55.21, -71.613, 63.734, 97.422, 14.668]
  MoveL 2886 to (239.62, 154.78, 50.44) mm, rotated rx 180 ry 0 rz 180 deg; joints [-62.778, 55.21, -71.613, 63.734, 97.422, 14.668]
  Call Extruder(652.24807)
  MoveL 2887 to (239.56, 154.97, 50.44) mm, rotated rx -180 ry 0 rz 180 deg; joints [-62.824, 55.221, -71.607, 63.777, 97.403, 14.66]
  MoveL 2888 to (239.56, 154.97, 50.44) mm, rotated rx -180 ry 0 rz 180 deg; joints [-62.824, 55.221, -71.607, 63.777, 97.403, 14.66]
  Call Extruder(652.36108)
  MoveL 2889 to (239.5, 155.15, 50.44) mm, rotated rx -180 ry 0 rz 180 deg; joints [-62.87, 55.232, -71.602, 63.821, 97.384, 14.651]
  MoveL 2890 to (239.5, 155.15, 50.44) mm, rotated rx -180 ry 0 rz 180 deg; joints [-62.87, 55.232, -71.602, 63.821, 97.384, 14.651]
  Call Extruder(652.47454)
  MoveL 2891 to (239.44, 155.34, 50.44) mm, rotated rx 180 ry 0 rz 180 deg; joints [-62.916, 55.242, -71.597, 63.864, 97.366, 14.643]
  MoveL 2892 to (239.44, 155.34, 50.44) mm, rotated rx 180 ry 0 rz 180 deg; joints [-62.916, 55.242, -71.597, 63.864, 97.366, 14.643]
  Call Extruder(652.62218)
  MoveL 2893 to (239.35, 155.58, 50.44) mm, rotated rx -180 ry 0 rz 180 deg; joints [-62.979, 55.255, -71.59, 63.923, 97.341, 14.633]
  MoveL 2894 to (239.35, 155.58, 50.44) mm, rotated rx -180 ry 0 rz 180 deg; joints [-62.979, 55.255, -71.59, 63.923, 97.341, 14.633]
  Call Extruder(652.80452)
  MoveL 2895 to (239.22, 155.87, 50.44) mm, rotated rx -180 ry 0 rz 180 deg; joints [-63.058, 55.271, -71.582, 63.997, 97.311, 14.621]
  MoveL 2896 to (239.22, 155.87, 50.44) mm, rotated rx -180 ry 0 rz 180 deg; joints [-63.058, 55.271, -71.582, 63.997, 97.311, 14.621]
  Call Extruder(652.98761)
  MoveL 2897 to (239.1, 156.17, 50.44) mm, rotated rx 180 ry 0 rz 180 deg; joints [-63.136, 55.287, -71.575, 64.07, 97.281, 14.609]
  MoveL 2898 to (239.1, 156.17, 50.44) mm, rotated rx 180 ry 0 rz 180 deg; joints [-63.136, 55.287, -71.575, 64.07, 97.281, 14.609]
  Call Extruder(653.14533)
  MoveL 2899 to (239, 156.42, 50.44) mm, rotated rx 180 ry 0 rz 180 deg; joints [-63.204, 55.3, -71.568, 64.135, 97.255, 14.6]
  MoveL 2900 to (239, 156.42, 50.44) mm, rotated rx 180 ry 0 rz 180 deg; joints [-63.204, 55.3, -71.568, 64.135, 97.255, 14.6]
  Call Extruder(653.30365)
  MoveL 2901 to (238.89, 156.66, 50.44) mm, rotated rx 180 ry 0 rz 180 deg; joints [-63.272, 55.313, -71.561, 64.198, 97.229, 14.59]
  MoveL 2902 to (238.89, 156.66, 50.44) mm, rotated rx 180 ry 0 rz 180 deg; joints [-63.272, 55.313, -71.561, 64.198, 97.229, 14.59]
  Call Extruder(653.48569)
  MoveL 2903 to (238.75, 156.94, 50.44) mm, rotated rx -180 ry 0 rz -180 deg; joints [-63.354, 55.327, -71.554, 64.276, 97.2, 14.581]
  MoveL 2904 to (238.75, 156.94, 50.44) mm, rotated rx -180 ry 0 rz -180 deg; joints [-63.354, 55.327, -71.554, 64.276, 97.2, 14.581]
  Call Extruder(653.69224)
  MoveL 2905 to (238.57, 157.25, 50.44) mm, rotated rx 180 ry 0 rz 180 deg; joints [-63.449, 55.342, -71.547, 64.367, 97.166, 14.573]
  MoveL 2906 to (238.57, 157.25, 50.44) mm, rotated rx 180 ry 0 rz 180 deg; joints [-63.449, 55.342, -71.547, 64.367, 97.166, 14.573]
  Call Extruder(653.89957)
  MoveL 2907 to (238.4, 157.55, 50.44) mm, rotated rx -180 ry 0 rz 180 deg; joints [-63.544, 55.357, -71.539, 64.457, 97.132, 14.564]
  MoveL 2908 to (238.4, 157.55, 50.44) mm, rotated rx -180 ry 0 rz 180 deg; joints [-63.544, 55.357, -71.539, 64.457, 97.132, 14.564]
  Call Extruder(654.10768)
  MoveL 2909 to (238.22, 157.85, 50.44) mm, rotated rx -180 ry 0 rz 180 deg; joints [-63.64, 55.371, -71.532, 64.547, 97.099, 14.556]
  MoveL 2910 to (238.22, 157.85, 50.44) mm, rotated rx -180 ry 0 rz 180 deg; joints [-63.64, 55.371, -71.532, 64.547, 97.099, 14.556]
  Call Extruder(654.22535)
  MoveL 2911 to (238.12, 158.02, 50.44) mm, rotated rx -180 ry 0 rz 180 deg; joints [-63.693, 55.38, -71.528, 64.598, 97.08, 14.551]
  MoveL 2912 to (238.12, 158.02, 50.44) mm, rotated rx -180 ry 0 rz 180 deg; joints [-63.693, 55.38, -71.528, 64.598, 97.08, 14.551]
  Call Extruder(654.55818)
  MoveL 2913 to (237.79, 158.48, 50.44) mm, rotated rx 180 ry 0 rz 180 deg; joints [-63.854, 55.399, -71.518, 64.752, 97.027, 14.543]
  MoveL 2914 to (237.79, 158.48, 50.44) mm, rotated rx 180 ry 0 rz 180 deg; joints [-63.854, 55.399, -71.518, 64.752, 97.027, 14.543]
  Call Extruder(654.89221)
  MoveL 2915 to (237.47, 158.93, 50.44) mm, rotated rx -180 ry 0 rz -180 deg; joints [-64.014, 55.419, -71.508, 64.904, 96.974, 14.535]
  MoveL 2916 to (237.47, 158.93, 50.44) mm, rotated rx -180 ry 0 rz -180 deg; joints [-64.014, 55.419, -71.508, 64.904, 96.974, 14.535]
  Call Extruder(655.05980)
  MoveL 2917 to (237.3, 159.15, 50.44) mm, rotated rx -180 ry 0 rz 180 deg; joints [-64.094, 55.429, -71.503, 64.98, 96.948, 14.53]
  Call Extruder(655.88912)
  MoveL 2918 to (236.39, 160.19, 50.44) mm, rotated rx 180 ry 0 rz 180 deg; joints [-64.505, 55.47, -71.482, 65.375, 96.819, 14.522]
  Call Extruder(656.52018)
  MoveL 2919 to (235.6, 160.89, 50.44) mm, rotated rx -180 ry 0 rz 180 deg; joints [-64.83, 55.492, -71.47, 65.688, 96.723, 14.529]
  MoveL 2920 to (235.6, 160.89, 50.44) mm, rotated rx -180 ry 0 rz 180 deg; joints [-64.83, 55.492, -71.47, 65.688, 96.723, 14.529]
  Call Extruder(656.71780)
  MoveL 2921 to (235.35, 161.1, 50.44) mm, rotated rx -180 ry 0 rz 180 deg; joints [-64.933, 55.498, -71.467, 65.787, 96.693, 14.531]
  Call Extruder(657.05182)
  MoveL 2922 to (234.9, 161.43, 50.44) mm, rotated rx -180 ry 0 rz 180 deg; joints [-65.109, 55.506, -71.463, 65.958, 96.644, 14.54]
  MoveL 2923 to (234.9, 161.43, 50.44) mm, rotated rx -180 ry 0 rz 180 deg; joints [-65.109, 55.506, -71.463, 65.958, 96.644, 14.54]
  Call Extruder(657.38465)
  MoveL 2924 to (234.45, 161.76, 50.44) mm, rotated rx -180 ry 0 rz 180 deg; joints [-65.285, 55.515, -71.458, 66.128, 96.595, 14.548]
  MoveL 2925 to (234.45, 161.76, 50.44) mm, rotated rx -180 ry 0 rz 180 deg; joints [-65.285, 55.515, -71.458, 66.128, 96.595, 14.548]
  Call Extruder(657.56385)
  MoveL 2926 to (234.21, 161.94, 50.44) mm, rotated rx 180 ry 0 rz -180 deg; joints [-65.381, 55.519, -71.456, 66.22, 96.568, 14.553]
  MoveL 2927 to (234.21, 161.94, 50.44) mm, rotated rx 180 ry 0 rz -180 deg; joints [-65.381, 55.519, -71.456, 66.22, 96.568, 14.553]
  Call Extruder(657.77197)
  MoveL 2928 to (233.9, 162.11, 50.44) mm, rotated rx 180 ry 0 rz 180 deg; joints [-65.493, 55.521, -71.455, 66.329, 96.539, 14.562]
  MoveL 2929 to (233.9, 162.11, 50.44) mm, rotated rx 180 ry 0 rz 180 deg; joints [-65.493, 55.521, -71.455, 66.329, 96.539, 14.562]
  Call Extruder(657.97930)
  MoveL 2930 to (233.6, 162.29, 50.44) mm, rotated rx 180 ry 0 rz -180 deg; joints [-65.605, 55.524, -71.453, 66.438, 96.509, 14.571]
  MoveL 2931 to (233.6, 162.29, 50.44) mm, rotated rx 180 ry 0 rz -180 deg; joints [-65.605, 55.524, -71.453, 66.438, 96.509, 14.571]
  Call Extruder(658.18586)
  MoveL 2932 to (233.29, 162.46, 50.44) mm, rotated rx 180 ry 0 rz 180 deg; joints [-65.718, 55.527, -71.452, 66.547, 96.479, 14.579]
  MoveL 2933 to (233.29, 162.46, 50.44) mm, rotated rx 180 ry 0 rz 180 deg; joints [-65.718, 55.527, -71.452, 66.547, 96.479, 14.579]
  Call Extruder(658.39164)
  MoveL 2934 to (232.99, 162.64, 50.44) mm, rotated rx 180 ry 0 rz 180 deg; joints [-65.83, 55.529, -71.451, 66.656, 96.449, 14.588]
  MoveL 2935 to (232.99, 162.64, 50.44) mm, rotated rx 180 ry 0 rz 180 deg; joints [-65.83, 55.529, -71.451, 66.656, 96.449, 14.588]
  Call Extruder(658.54991)
  MoveL 2936 to (232.74, 162.74, 50.44) mm, rotated rx -180 ry 0 rz 180 deg; joints [-65.917, 55.529, -71.451, 66.741, 96.427, 14.598]
  MoveL 2937 to (232.74, 162.74, 50.44) mm, rotated rx -180 ry 0 rz 180 deg; joints [-65.917, 55.529, -71.451, 66.741, 96.427, 14.598]
  Call Extruder(658.70759)
  MoveL 2938 to (232.49, 162.85, 50.44) mm, rotated rx 180 ry 0 rz -180 deg; joints [-66.004, 55.529, -71.451, 66.826, 96.405, 14.608]
  MoveL 2939 to (232.49, 162.85, 50.44) mm, rotated rx 180 ry 0 rz -180 deg; joints [-66.004, 55.529, -71.451, 66.826, 96.405, 14.608]
  Call Extruder(658.87768)
  MoveL 2940 to (232.22, 162.96, 50.44) mm, rotated rx 180 ry 0 rz 180 deg; joints [-66.099, 55.528, -71.451, 66.918, 96.382, 14.619]
  MoveL 2941 to (232.22, 162.96, 50.44) mm, rotated rx 180 ry 0 rz 180 deg; joints [-66.099, 55.528, -71.451, 66.918, 96.382, 14.619]
  Call Extruder(659.06004)
  MoveL 2942 to (231.93, 163.09, 50.44) mm, rotated rx -180 ry 0 rz 180 deg; joints [-66.2, 55.528, -71.451, 67.017, 96.357, 14.63]
  MoveL 2943 to (231.93, 163.09, 50.44) mm, rotated rx -180 ry 0 rz 180 deg; joints [-66.2, 55.528, -71.451, 67.017, 96.357, 14.63]
  Call Extruder(659.24164)
  MoveL 2944 to (231.64, 163.21, 50.44) mm, rotated rx 180 ry 0 rz 180 deg; joints [-66.302, 55.527, -71.452, 67.116, 96.331, 14.642]
  MoveL 2945 to (231.64, 163.21, 50.44) mm, rotated rx 180 ry 0 rz 180 deg; joints [-66.302, 55.527, -71.452, 67.116, 96.331, 14.642]
  Call Extruder(659.35509)
  MoveL 2946 to (231.45, 163.27, 50.44) mm, rotated rx 180 ry 0 rz -180 deg; joints [-66.365, 55.526, -71.452, 67.178, 96.316, 14.651]
  MoveL 2947 to (231.45, 163.27, 50.44) mm, rotated rx 180 ry 0 rz -180 deg; joints [-66.365, 55.526, -71.452, 67.178, 96.316, 14.651]
  Call Extruder(659.46809)
  MoveL 2948 to (231.26, 163.33, 50.44) mm, rotated rx 180 ry 0 rz 180 deg; joints [-66.428, 55.524, -71.453, 67.24, 96.301, 14.66]
  MoveL 2949 to (231.26, 163.33, 50.44) mm, rotated rx 180 ry 0 rz 180 deg; joints [-66.428, 55.524, -71.453, 67.24, 96.301, 14.66]
  Call Extruder(659.58064)
  MoveL 2950 to (231.07, 163.39, 50.44) mm, rotated rx -180 ry 0 rz 180 deg; joints [-66.492, 55.523, -71.454, 67.302, 96.286, 14.668]
  MoveL 2951 to (231.07, 163.39, 50.44) mm, rotated rx -180 ry 0 rz 180 deg; joints [-66.492, 55.523, -71.454, 67.302, 96.286, 14.668]
  Call Extruder(659.69275)
  MoveL 2952 to (230.88, 163.45, 50.44) mm, rotated rx -180 ry 0 rz -180 deg; joints [-66.555, 55.521, -71.455, 67.364, 96.27, 14.677]
  MoveL 2953 to (230.88, 163.45, 50.44) mm, rotated rx -180 ry 0 rz -180 deg; joints [-66.555, 55.521, -71.455, 67.364, 96.27, 14.677]
  Call Extruder(659.80442)
  MoveL 2954 to (230.69, 163.51, 50.44) mm, rotated rx -180 ry 0 rz -180 deg; joints [-66.619, 55.52, -71.455, 67.426, 96.255, 14.686]
  MoveL 2955 to (230.69, 163.51, 50.44) mm, rotated rx -180 ry 0 rz -180 deg; joints [-66.619, 55.52, -71.455, 67.426, 96.255, 14.686]
  Call Extruder(659.93552)
  MoveL 2956 to (230.47, 163.58, 50.44) mm, rotated rx -180 ry 0 rz 180 deg; joints [-66.694, 55.518, -71.457, 67.499, 96.237, 14.697]
  MoveL 2957 to (230.47, 163.58, 50.44) mm, rotated rx -180 ry 0 rz 180 deg; joints [-66.694, 55.518, -71.457, 67.499, 96.237, 14.697]
  Call Extruder(660.06605)
  MoveL 2958 to (230.25, 163.65, 50.44) mm, rotated rx -180 ry 0 rz -180 deg; joints [-66.768, 55.516, -71.458, 67.572, 96.22, 14.707]
  MoveL 2959 to (230.25, 163.65, 50.44) mm, rotated rx -180 ry 0 rz -180 deg; joints [-66.768, 55.516, -71.458, 67.572, 96.22, 14.707]
  Call Extruder(660.19601)
  MoveL 2960 to (230.02, 163.72, 50.44) mm, rotated rx -180 ry 0 rz 180 deg; joints [-66.843, 55.514, -71.459, 67.645, 96.202, 14.718]
  MoveL 2961 to (230.02, 163.72, 50.44) mm, rotated rx -180 ry 0 rz 180 deg; joints [-66.843, 55.514, -71.459, 67.645, 96.202, 14.718]
  Call Extruder(660.32541)
  MoveL 2962 to (229.8, 163.78, 50.44) mm, rotated rx -180 ry 0 rz 180 deg; joints [-66.918, 55.512, -71.46, 67.718, 96.184, 14.729]
  MoveL 2963 to (229.8, 163.78, 50.44) mm, rotated rx -180 ry 0 rz 180 deg; joints [-66.918, 55.512, -71.46, 67.718, 96.184, 14.729]
  Call Extruder(660.44739)
  MoveL 2964 to (229.59, 163.84, 50.44) mm, rotated rx -180 ry 0 rz -180 deg; joints [-66.988, 55.51, -71.461, 67.787, 96.167, 14.739]
  MoveL 2965 to (229.59, 163.84, 50.44) mm, rotated rx -180 ry 0 rz -180 deg; joints [-66.988, 55.51, -71.461, 67.787, 96.167, 14.739]
  Call Extruder(660.56223)
  MoveL 2966 to (229.38, 163.88, 50.44) mm, rotated rx -180 ry 0 rz 180 deg; joints [-67.054, 55.507, -71.462, 67.851, 96.152, 14.75]
  MoveL 2967 to (229.38, 163.88, 50.44) mm, rotated rx -180 ry 0 rz 180 deg; joints [-67.054, 55.507, -71.462, 67.851, 96.152, 14.75]
  Call Extruder(660.67663)
  MoveL 2968 to (229.18, 163.93, 50.44) mm, rotated rx -180 ry 0 rz -180 deg; joints [-67.12, 55.504, -71.464, 67.916, 96.137, 14.761]
  MoveL 2969 to (229.18, 163.93, 50.44) mm, rotated rx -180 ry 0 rz -180 deg; joints [-67.12, 55.504, -71.464, 67.916, 96.137, 14.761]
  Call Extruder(660.79057)
  MoveL 2970 to (228.97, 163.97, 50.44) mm, rotated rx -180 ry 0 rz 180 deg; joints [-67.187, 55.501, -71.465, 67.981, 96.122, 14.772]
  MoveL 2971 to (228.97, 163.97, 50.44) mm, rotated rx -180 ry 0 rz 180 deg; joints [-67.187, 55.501, -71.465, 67.981, 96.122, 14.772]
  Call Extruder(660.90406)
  MoveL 2972 to (228.77, 164.02, 50.44) mm, rotated rx 180 ry 0 rz 180 deg; joints [-67.253, 55.498, -71.467, 68.046, 96.106, 14.783]
  MoveL 2973 to (228.77, 164.02, 50.44) mm, rotated rx 180 ry 0 rz 180 deg; joints [-67.253, 55.498, -71.467, 68.046, 96.106, 14.783]
  Call Extruder(661.04134)
  MoveL 2974 to (228.52, 164.07, 50.44) mm, rotated rx -180 ry 0 rz 180 deg; joints [-67.333, 55.494, -71.469, 68.124, 96.088, 14.797]
  MoveL 2975 to (228.52, 164.07, 50.44) mm, rotated rx -180 ry 0 rz 180 deg; joints [-67.333, 55.494, -71.469, 68.124, 96.088, 14.797]
  Call Extruder(661.17802)
  MoveL 2976 to (228.27, 164.12, 50.44) mm, rotated rx -180 ry 0 rz -180 deg; joints [-67.413, 55.491, -71.471, 68.203, 96.07, 14.81]
  MoveL 2977 to (228.27, 164.12, 50.44) mm, rotated rx -180 ry 0 rz -180 deg; joints [-67.413, 55.491, -71.471, 68.203, 96.07, 14.81]
  Call Extruder(661.31408)
  MoveL 2978 to (228.02, 164.17, 50.44) mm, rotated rx -180 ry 0 rz 180 deg; joints [-67.494, 55.487, -71.473, 68.281, 96.051, 14.824]
  MoveL 2979 to (228.02, 164.17, 50.44) mm, rotated rx -180 ry 0 rz 180 deg; joints [-67.494, 55.487, -71.473, 68.281, 96.051, 14.824]
  Call Extruder(661.44953)
  MoveL 2980 to (227.77, 164.22, 50.44) mm, rotated rx -180 ry 0 rz 180 deg; joints [-67.574, 55.483, -71.475, 68.36, 96.033, 14.838]
  MoveL 2981 to (227.77, 164.22, 50.44) mm, rotated rx -180 ry 0 rz 180 deg; joints [-67.574, 55.483, -71.475, 68.36, 96.033, 14.838]
  Call Extruder(661.58438)
  MoveL 2982 to (227.52, 164.27, 50.44) mm, rotated rx 180 ry 0 rz 180 deg; joints [-67.654, 55.479, -71.477, 68.439, 96.014, 14.851]
  MoveL 2983 to (227.52, 164.27, 50.44) mm, rotated rx 180 ry 0 rz 180 deg; joints [-67.654, 55.479, -71.477, 68.439, 96.014, 14.851]
  Call Extruder(661.71861)
  MoveL 2984 to (227.27, 164.32, 50.44) mm, rotated rx 180 ry 0 rz 180 deg; joints [-67.735, 55.476, -71.478, 68.517, 95.996, 14.864]
  MoveL 2985 to (227.27, 164.32, 50.44) mm, rotated rx 180 ry 0 rz 180 deg; joints [-67.735, 55.476, -71.478, 68.517, 95.996, 14.864]
  Call Extruder(661.85223)
  MoveL 2986 to (227.02, 164.36, 50.44) mm, rotated rx -180 ry 0 rz 180 deg; joints [-67.815, 55.472, -71.48, 68.596, 95.977, 14.878]
  MoveL 2987 to (227.02, 164.36, 50.44) mm, rotated rx -180 ry 0 rz 180 deg; joints [-67.815, 55.472, -71.48, 68.596, 95.977, 14.878]
  Call Extruder(662.01433)
  MoveL 2988 to (226.72, 164.41, 50.44) mm, rotated rx -180 ry 0 rz 180 deg; joints [-67.912, 55.467, -71.483, 68.692, 95.955, 14.895]
  MoveL 2989 to (226.72, 164.41, 50.44) mm, rotated rx -180 ry 0 rz 180 deg; joints [-67.912, 55.467, -71.483, 68.692, 95.955, 14.895]
  Call Extruder(662.17571)
  MoveL 2990 to (226.41, 164.46, 50.44) mm, rotated rx 180 ry 0 rz 180 deg; joints [-68.01, 55.461, -71.486, 68.787, 95.933, 14.912]
  MoveL 2991 to (226.41, 164.46, 50.44) mm, rotated rx 180 ry 0 rz 180 deg; joints [-68.01, 55.461, -71.486, 68.787, 95.933, 14.912]
  Call Extruder(662.33636)
  MoveL 2992 to (226.11, 164.51, 50.44) mm, rotated rx -180 ry 0 rz 180 deg; joints [-68.107, 55.456, -71.488, 68.883, 95.911, 14.93]
  MoveL 2993 to (226.11, 164.51, 50.44) mm, rotated rx -180 ry 0 rz 180 deg; joints [-68.107, 55.456, -71.488, 68.883, 95.911, 14.93]
  Call Extruder(662.49628)
  MoveL 2994 to (225.8, 164.56, 50.44) mm, rotated rx -180 ry 0 rz 180 deg; joints [-68.205, 55.451, -71.491, 68.978, 95.888, 14.947]
  MoveL 2995 to (225.8, 164.56, 50.44) mm, rotated rx -180 ry 0 rz 180 deg; joints [-68.205, 55.451, -71.491, 68.978, 95.888, 14.947]
  Call Extruder(662.65547)
  MoveL 2996 to (225.5, 164.61, 50.44) mm, rotated rx -180 ry 0 rz 180 deg; joints [-68.303, 55.446, -71.494, 69.074, 95.866, 14.964]
  MoveL 2997 to (225.5, 164.61, 50.44) mm, rotated rx -180 ry 0 rz 180 deg; joints [-68.303, 55.446, -71.494, 69.074, 95.866, 14.964]
  Call Extruder(662.81393)
  MoveL 2998 to (225.19, 164.66, 50.44) mm, rotated rx 180 ry 0 rz 180 deg; joints [-68.4, 55.441, -71.496, 69.169, 95.843, 14.981]
  MoveL 2999 to (225.19, 164.66, 50.44) mm, rotated rx 180 ry 0 rz 180 deg; joints [-68.4, 55.441, -71.496, 69.169, 95.843, 14.981]
  Call Extruder(663.01281)
  MoveL 3000 to (224.8, 164.7, 50.44) mm, rotated rx -180 ry 0 rz 180 deg; joints [-68.522, 55.433, -71.5, 69.289, 95.816, 15.003]
  MoveL 3001 to (224.8, 164.7, 50.44) mm, rotated rx -180 ry 0 rz 180 deg; joints [-68.522, 55.433, -71.5, 69.289, 95.816, 15.003]
  Call Extruder(663.21082)
  MoveL 3002 to (224.42, 164.75, 50.44) mm, rotated rx -180 ry 0 rz -180 deg; joints [-68.645, 55.426, -71.504, 69.409, 95.788, 15.026]
  MoveL 3003 to (224.42, 164.75, 50.44) mm, rotated rx -180 ry 0 rz -180 deg; joints [-68.645, 55.426, -71.504, 69.409, 95.788, 15.026]
  Call Extruder(663.40796)
  MoveL 3004 to (224.03, 164.79, 50.44) mm, rotated rx -180 ry 0 rz 180 deg; joints [-68.767, 55.418, -71.508, 69.528, 95.76, 15.048]
  MoveL 3005 to (224.03, 164.79, 50.44) mm, rotated rx -180 ry 0 rz 180 deg; joints [-68.767, 55.418, -71.508, 69.528, 95.76, 15.048]
  Call Extruder(663.60423)
  MoveL 3006 to (223.64, 164.84, 50.44) mm, rotated rx 180 ry 0 rz -180 deg; joints [-68.89, 55.411, -71.512, 69.648, 95.732, 15.071]
  MoveL 3007 to (223.64, 164.84, 50.44) mm, rotated rx 180 ry 0 rz -180 deg; joints [-68.89, 55.411, -71.512, 69.648, 95.732, 15.071]
  Call Extruder(663.84990)
  MoveL 3008 to (223.15, 164.89, 50.44) mm, rotated rx 180 ry 0 rz 180 deg; joints [-69.043, 55.401, -71.517, 69.798, 95.698, 15.1]
  MoveL 3009 to (223.15, 164.89, 50.44) mm, rotated rx 180 ry 0 rz 180 deg; joints [-69.043, 55.401, -71.517, 69.798, 95.698, 15.1]
  Call Extruder(664.14459)
  MoveL 3010 to (222.56, 164.93, 50.44) mm, rotated rx -180 ry 0 rz 180 deg; joints [-69.227, 55.388, -71.523, 69.979, 95.656, 15.136]
  MoveL 3011 to (222.56, 164.93, 50.44) mm, rotated rx -180 ry 0 rz 180 deg; joints [-69.227, 55.388, -71.523, 69.979, 95.656, 15.136]
  Call Extruder(664.43795)
  MoveL 3012 to (221.97, 164.98, 50.44) mm, rotated rx -180 ry 0 rz -180 deg; joints [-69.411, 55.376, -71.53, 70.16, 95.615, 15.171]
  MoveL 3013 to (221.97, 164.98, 50.44) mm, rotated rx -180 ry 0 rz -180 deg; joints [-69.411, 55.376, -71.53, 70.16, 95.615, 15.171]
  Call Extruder(664.87126)
  MoveL 3014 to (221.1, 165.02, 50.44) mm, rotated rx -180 ry 0 rz 180 deg; joints [-69.684, 55.356, -71.54, 70.426, 95.553, 15.225]
  MoveL 3015 to (221.1, 165.02, 50.44) mm, rotated rx -180 ry 0 rz 180 deg; joints [-69.684, 55.356, -71.54, 70.426, 95.553, 15.225]
  Call Extruder(665.44342)
  MoveL 3016 to (219.94, 165.07, 50.44) mm, rotated rx 180 ry 0 rz 180 deg; joints [-70.044, 55.329, -71.553, 70.78, 95.472, 15.297]
  MoveL 3017 to (219.94, 165.07, 50.44) mm, rotated rx 180 ry 0 rz 180 deg; joints [-70.044, 55.329, -71.553, 70.78, 95.472, 15.297]
  Call Extruder(665.87130)
  MoveL 3018 to (219.06, 165.09, 50.44) mm, rotated rx 180 ry 0 rz -180 deg; joints [-70.315, 55.308, -71.564, 71.045, 95.411, 15.352]
  Call Extruder(782.51995)
  MoveL 3019 to (-19.06, 165.09, 50.44) mm, rotated rx -180 ry 0 rz 180 deg; joints [-137.325, 59.836, -68.062, 137.03, 83.961, 5.597]
  MoveL 3020 to (-19.06, 165.09, 50.44) mm, rotated rx -180 ry 0 rz 180 deg; joints [-137.325, 59.836, -68.062, 137.03, 83.961, 5.597]
  Call Extruder(783.23557)
  MoveL 3021 to (-20.52, 165.05, 50.44) mm, rotated rx 180 ry 0 rz 180 deg; joints [-137.563, 59.895, -67.995, 137.277, 84.031, 5.486]
  MoveL 3022 to (-20.52, 165.05, 50.44) mm, rotated rx 180 ry 0 rz 180 deg; joints [-137.563, 59.895, -67.995, 137.277, 84.031, 5.486]
  Call Extruder(783.81031)
  MoveL 3023 to (-21.68, 165, 50.44) mm, rotated rx -180 ry 0 rz -180 deg; joints [-137.754, 59.941, -67.94, 137.475, 84.087, 5.397]
  MoveL 3024 to (-21.68, 165, 50.44) mm, rotated rx -180 ry 0 rz -180 deg; joints [-137.754, 59.941, -67.94, 137.475, 84.087, 5.397]
  Call Extruder(784.10367)
  MoveL 3025 to (-22.27, 164.96, 50.44) mm, rotated rx -180 ry 0 rz 180 deg; joints [-137.855, 59.963, -67.914, 137.579, 84.114, 5.354]
  MoveL 3026 to (-22.27, 164.96, 50.44) mm, rotated rx -180 ry 0 rz 180 deg; joints [-137.855, 59.963, -67.914, 137.579, 84.114, 5.354]
  Call Extruder(784.39837)
  MoveL 3027 to (-22.86, 164.91, 50.44) mm, rotated rx 180 ry 0 rz 180 deg; joints [-137.955, 59.986, -67.887, 137.683, 84.141, 5.31]
  MoveL 3028 to (-22.86, 164.91, 50.44) mm, rotated rx 180 ry 0 rz 180 deg; joints [-137.955, 59.986, -67.887, 137.683, 84.141, 5.31]
  Call Extruder(784.69439)
  MoveL 3029 to (-23.45, 164.86, 50.44) mm, rotated rx 180 ry 0 rz 180 deg; joints [-138.054, 60.009, -67.861, 137.786, 84.168, 5.267]
  MoveL 3030 to (-23.45, 164.86, 50.44) mm, rotated rx 180 ry 0 rz 180 deg; joints [-138.054, 60.009, -67.861, 137.786, 84.168, 5.267]
  Call Extruder(784.89067)
  MoveL 3031 to (-23.83, 164.82, 50.44) mm, rotated rx 180 ry 0 rz 180 deg; joints [-138.122, 60.023, -67.844, 137.856, 84.185, 5.239]
  MoveL 3032 to (-23.83, 164.82, 50.44) mm, rotated rx 180 ry 0 rz 180 deg; joints [-138.122, 60.023, -67.844, 137.856, 84.185, 5.239]
  Call Extruder(785.08781)
  MoveL 3033 to (-24.22, 164.77, 50.44) mm, rotated rx -180 ry 0 rz 180 deg; joints [-138.19, 60.037, -67.827, 137.926, 84.202, 5.211]
  MoveL 3034 to (-24.22, 164.77, 50.44) mm, rotated rx -180 ry 0 rz 180 deg; joints [-138.19, 60.037, -67.827, 137.926, 84.202, 5.211]
  Call Extruder(785.28582)
  MoveL 3035 to (-24.61, 164.72, 50.44) mm, rotated rx -180 ry 0 rz -180 deg; joints [-138.258, 60.052, -67.809, 137.996, 84.219, 5.183]
  MoveL 3036 to (-24.61, 164.72, 50.44) mm, rotated rx -180 ry 0 rz -180 deg; joints [-138.258, 60.052, -67.809, 137.996, 84.219, 5.183]
  Call Extruder(785.48469)
  MoveL 3037 to (-25, 164.68, 50.44) mm, rotated rx -180 ry 0 rz 180 deg; joints [-138.325, 60.066, -67.792, 138.066, 84.237, 5.155]
  MoveL 3038 to (-25, 164.68, 50.44) mm, rotated rx -180 ry 0 rz 180 deg; joints [-138.325, 60.066, -67.792, 138.066, 84.237, 5.155]
  Call Extruder(785.66377)
  MoveL 3039 to (-25.34, 164.63, 50.44) mm, rotated rx -180 ry 0 rz -180 deg; joints [-138.387, 60.078, -67.777, 138.129, 84.252, 5.13]
  MoveL 3040 to (-25.34, 164.63, 50.44) mm, rotated rx -180 ry 0 rz -180 deg; joints [-138.387, 60.078, -67.777, 138.129, 84.252, 5.13]
  Call Extruder(785.82297)
  MoveL 3041 to (-25.65, 164.58, 50.44) mm, rotated rx -180 ry 0 rz 180 deg; joints [-138.442, 60.089, -67.764, 138.186, 84.264, 5.108]
  MoveL 3042 to (-25.65, 164.58, 50.44) mm, rotated rx -180 ry 0 rz 180 deg; joints [-138.442, 60.089, -67.764, 138.186, 84.264, 5.108]
  Call Extruder(785.98289)
  MoveL 3043 to (-25.96, 164.53, 50.44) mm, rotated rx -180 ry 0 rz -180 deg; joints [-138.497, 60.1, -67.751, 138.243, 84.277, 5.087]
  MoveL 3044 to (-25.96, 164.53, 50.44) mm, rotated rx -180 ry 0 rz -180 deg; joints [-138.497, 60.1, -67.751, 138.243, 84.277, 5.087]
  Call Extruder(786.14354)
  MoveL 3045 to (-26.26, 164.49, 50.44) mm, rotated rx 180 ry 0 rz 180 deg; joints [-138.552, 60.111, -67.738, 138.3, 84.29, 5.066]
  MoveL 3046 to (-26.26, 164.49, 50.44) mm, rotated rx 180 ry 0 rz 180 deg; joints [-138.552, 60.111, -67.738, 138.3, 84.29, 5.066]
  Call Extruder(786.30492)
  MoveL 3047 to (-26.57, 164.44, 50.44) mm, rotated rx -180 ry 0 rz 180 deg; joints [-138.607, 60.122, -67.725, 138.356, 84.303, 5.044]
  MoveL 3048 to (-26.57, 164.44, 50.44) mm, rotated rx -180 ry 0 rz 180 deg; joints [-138.607, 60.122, -67.725, 138.356, 84.303, 5.044]
  Call Extruder(786.46703)
  MoveL 3049 to (-26.87, 164.39, 50.44) mm, rotated rx 180 ry 0 rz 180 deg; joints [-138.662, 60.132, -67.712, 138.413, 84.317, 5.023]
  MoveL 3050 to (-26.87, 164.39, 50.44) mm, rotated rx 180 ry 0 rz 180 deg; joints [-138.662, 60.132, -67.712, 138.413, 84.317, 5.023]
  Call Extruder(786.61523)
  MoveL 3051 to (-27.15, 164.34, 50.44) mm, rotated rx -180 ry 0 rz 180 deg; joints [-138.713, 60.142, -67.7, 138.465, 84.328, 5.003]
  MoveL 3052 to (-27.15, 164.34, 50.44) mm, rotated rx -180 ry 0 rz 180 deg; joints [-138.713, 60.142, -67.7, 138.465, 84.328, 5.003]
  Call Extruder(786.74946)
  MoveL 3053 to (-27.4, 164.29, 50.44) mm, rotated rx -180 ry 0 rz -180 deg; joints [-138.759, 60.15, -67.69, 138.513, 84.338, 4.986]
  MoveL 3054 to (-27.4, 164.29, 50.44) mm, rotated rx -180 ry 0 rz -180 deg; joints [-138.759, 60.15, -67.69, 138.513, 84.338, 4.986]
  Call Extruder(786.88430)
  MoveL 3055 to (-27.65, 164.24, 50.44) mm, rotated rx -180 ry 0 rz 180 deg; joints [-138.806, 60.159, -67.679, 138.56, 84.348, 4.969]
  MoveL 3056 to (-27.65, 164.24, 50.44) mm, rotated rx -180 ry 0 rz 180 deg; joints [-138.806, 60.159, -67.679, 138.56, 84.348, 4.969]
  Call Extruder(787.01975)
  MoveL 3057 to (-27.9, 164.19, 50.44) mm, rotated rx -180 ry 0 rz 180 deg; joints [-138.852, 60.167, -67.669, 138.608, 84.358, 4.952]
  MoveL 3058 to (-27.9, 164.19, 50.44) mm, rotated rx -180 ry 0 rz 180 deg; joints [-138.852, 60.167, -67.669, 138.608, 84.358, 4.952]
  Call Extruder(787.15582)
  MoveL 3059 to (-28.15, 164.14, 50.44) mm, rotated rx -180 ry 0 rz -180 deg; joints [-138.898, 60.176, -67.658, 138.655, 84.368, 4.935]
  MoveL 3060 to (-28.15, 164.14, 50.44) mm, rotated rx -180 ry 0 rz -180 deg; joints [-138.898, 60.176, -67.658, 138.655, 84.368, 4.935]
  Call Extruder(787.29249)
  MoveL 3061 to (-28.4, 164.09, 50.44) mm, rotated rx 180 ry 0 rz 180 deg; joints [-138.944, 60.184, -67.648, 138.703, 84.379, 4.918]
  MoveL 3062 to (-28.4, 164.09, 50.44) mm, rotated rx 180 ry 0 rz 180 deg; joints [-138.944, 60.184, -67.648, 138.703, 84.379, 4.918]
  Call Extruder(787.42977)
  MoveL 3063 to (-28.64, 164.04, 50.44) mm, rotated rx -180 ry 0 rz -180 deg; joints [-138.99, 60.193, -67.638, 138.75, 84.389, 4.901]
  MoveL 3064 to (-28.64, 164.04, 50.44) mm, rotated rx -180 ry 0 rz -180 deg; joints [-138.99, 60.193, -67.638, 138.75, 84.389, 4.901]
  Call Extruder(787.55544)
  MoveL 3065 to (-28.87, 164, 50.44) mm, rotated rx -180 ry 0 rz 180 deg; joints [-139.032, 60.2, -67.628, 138.793, 84.398, 4.885]
  MoveL 3066 to (-28.87, 164, 50.44) mm, rotated rx -180 ry 0 rz 180 deg; joints [-139.032, 60.2, -67.628, 138.793, 84.398, 4.885]
  Call Extruder(787.66938)
  MoveL 3067 to (-29.08, 163.95, 50.44) mm, rotated rx -180 ry 0 rz 180 deg; joints [-139.071, 60.207, -67.62, 138.833, 84.406, 4.872]
  MoveL 3068 to (-29.08, 163.95, 50.44) mm, rotated rx -180 ry 0 rz 180 deg; joints [-139.071, 60.207, -67.62, 138.833, 84.406, 4.872]
  Call Extruder(787.78378)
  MoveL 3069 to (-29.28, 163.91, 50.44) mm, rotated rx 180 ry 0 rz -180 deg; joints [-139.109, 60.214, -67.611, 138.872, 84.415, 4.858]
  MoveL 3070 to (-29.28, 163.91, 50.44) mm, rotated rx 180 ry 0 rz -180 deg; joints [-139.109, 60.214, -67.611, 138.872, 84.415, 4.858]
  Call Extruder(787.89862)
  MoveL 3071 to (-29.48, 163.86, 50.44) mm, rotated rx -180 ry 0 rz 180 deg; joints [-139.147, 60.221, -67.603, 138.911, 84.423, 4.844]
  MoveL 3072 to (-29.48, 163.86, 50.44) mm, rotated rx -180 ry 0 rz 180 deg; joints [-139.147, 60.221, -67.603, 138.911, 84.423, 4.844]
  Call Extruder(788.01392)
  MoveL 3073 to (-29.69, 163.82, 50.44) mm, rotated rx -180 ry 0 rz -180 deg; joints [-139.186, 60.228, -67.594, 138.951, 84.431, 4.83]
  MoveL 3074 to (-29.69, 163.82, 50.44) mm, rotated rx -180 ry 0 rz -180 deg; joints [-139.186, 60.228, -67.594, 138.951, 84.431, 4.83]
  Call Extruder(788.14332)
  MoveL 3075 to (-29.91, 163.75, 50.44) mm, rotated rx -180 ry 0 rz 180 deg; joints [-139.231, 60.234, -67.586, 138.997, 84.439, 4.816]
  MoveL 3076 to (-29.91, 163.75, 50.44) mm, rotated rx -180 ry 0 rz 180 deg; joints [-139.231, 60.234, -67.586, 138.997, 84.439, 4.816]
  Call Extruder(788.27328)
  MoveL 3077 to (-30.14, 163.68, 50.44) mm, rotated rx 180 ry 0 rz 180 deg; joints [-139.276, 60.241, -67.578, 139.043, 84.447, 4.801]
  MoveL 3078 to (-30.14, 163.68, 50.44) mm, rotated rx 180 ry 0 rz 180 deg; joints [-139.276, 60.241, -67.578, 139.043, 84.447, 4.801]
  Call Extruder(788.40380)
  MoveL 3079 to (-30.36, 163.61, 50.44) mm, rotated rx -180 ry 0 rz -180 deg; joints [-139.321, 60.248, -67.569, 139.089, 84.454, 4.787]
  MoveL 3080 to (-30.36, 163.61, 50.44) mm, rotated rx -180 ry 0 rz -180 deg; joints [-139.321, 60.248, -67.569, 139.089, 84.454, 4.787]
  Call Extruder(788.53489)
  MoveL 3081 to (-30.58, 163.55, 50.44) mm, rotated rx -180 ry 0 rz 180 deg; joints [-139.366, 60.255, -67.561, 139.135, 84.462, 4.773]
  MoveL 3082 to (-30.58, 163.55, 50.44) mm, rotated rx -180 ry 0 rz 180 deg; joints [-139.366, 60.255, -67.561, 139.135, 84.462, 4.773]
  Call Extruder(788.65654)
  MoveL 3083 to (-30.79, 163.48, 50.44) mm, rotated rx -180 ry 0 rz 180 deg; joints [-139.408, 60.261, -67.553, 139.178, 84.469, 4.759]
  MoveL 3084 to (-30.79, 163.48, 50.44) mm, rotated rx -180 ry 0 rz 180 deg; joints [-139.408, 60.261, -67.553, 139.178, 84.469, 4.759]
  Call Extruder(788.76865)
  MoveL 3085 to (-30.98, 163.42, 50.44) mm, rotated rx -180 ry 0 rz 180 deg; joints [-139.446, 60.266, -67.546, 139.217, 84.475, 4.748]
  MoveL 3086 to (-30.98, 163.42, 50.44) mm, rotated rx -180 ry 0 rz 180 deg; joints [-139.446, 60.266, -67.546, 139.217, 84.475, 4.748]
  Call Extruder(788.88121)
  MoveL 3087 to (-31.17, 163.36, 50.44) mm, rotated rx -180 ry 0 rz -180 deg; joints [-139.485, 60.272, -67.539, 139.256, 84.482, 4.735]
  MoveL 3088 to (-31.17, 163.36, 50.44) mm, rotated rx -180 ry 0 rz -180 deg; joints [-139.485, 60.272, -67.539, 139.256, 84.482, 4.735]
  Call Extruder(788.99421)
  MoveL 3089 to (-31.35, 163.3, 50.44) mm, rotated rx 180 ry 0 rz 180 deg; joints [-139.523, 60.278, -67.532, 139.295, 84.488, 4.724]
  MoveL 3090 to (-31.35, 163.3, 50.44) mm, rotated rx 180 ry 0 rz 180 deg; joints [-139.523, 60.278, -67.532, 139.295, 84.488, 4.724]
  Call Extruder(789.10766)
  MoveL 3091 to (-31.54, 163.24, 50.44) mm, rotated rx 180 ry 0 rz 180 deg; joints [-139.562, 60.283, -67.525, 139.335, 84.495, 4.712]
  MoveL 3092 to (-31.54, 163.24, 50.44) mm, rotated rx 180 ry 0 rz 180 deg; joints [-139.562, 60.283, -67.525, 139.335, 84.495, 4.712]
  Call Extruder(789.25531)
  MoveL 3093 to (-31.78, 163.15, 50.44) mm, rotated rx -180 ry 0 rz 180 deg; joints [-139.613, 60.29, -67.516, 139.387, 84.502, 4.697]
  MoveL 3094 to (-31.78, 163.15, 50.44) mm, rotated rx -180 ry 0 rz 180 deg; joints [-139.613, 60.29, -67.516, 139.387, 84.502, 4.697]
  Call Extruder(789.43766)
  MoveL 3095 to (-32.08, 163.02, 50.44) mm, rotated rx -180 ry 0 rz 180 deg; joints [-139.677, 60.298, -67.507, 139.452, 84.51, 4.679]
  MoveL 3096 to (-32.08, 163.02, 50.44) mm, rotated rx -180 ry 0 rz 180 deg; joints [-139.677, 60.298, -67.507, 139.452, 84.51, 4.679]
  Call Extruder(789.62078)
  MoveL 3097 to (-32.37, 162.91, 50.44) mm, rotated rx -180 ry 0 rz -180 deg; joints [-139.741, 60.305, -67.497, 139.517, 84.518, 4.662]
  MoveL 3098 to (-32.37, 162.91, 50.44) mm, rotated rx -180 ry 0 rz -180 deg; joints [-139.741, 60.305, -67.497, 139.517, 84.518, 4.662]
  Call Extruder(789.77845)
  MoveL 3099 to (-32.62, 162.8, 50.44) mm, rotated rx -180 ry 0 rz 180 deg; joints [-139.796, 60.312, -67.488, 139.573, 84.525, 4.647]
  MoveL 3100 to (-32.62, 162.8, 50.44) mm, rotated rx -180 ry 0 rz 180 deg; joints [-139.796, 60.312, -67.488, 139.573, 84.525, 4.647]
  Call Extruder(789.93673)
  MoveL 3101 to (-32.86, 162.69, 50.44) mm, rotated rx -180 ry 0 rz 180 deg; joints [-139.851, 60.319, -67.48, 139.629, 84.532, 4.632]
  MoveL 3102 to (-32.86, 162.69, 50.44) mm, rotated rx -180 ry 0 rz 180 deg; joints [-139.851, 60.319, -67.48, 139.629, 84.532, 4.632]
  Call Extruder(790.11874)
  MoveL 3103 to (-33.14, 162.55, 50.44) mm, rotated rx 180 ry 0 rz 180 deg; joints [-139.916, 60.325, -67.472, 139.696, 84.538, 4.616]
  MoveL 3104 to (-33.14, 162.55, 50.44) mm, rotated rx 180 ry 0 rz 180 deg; joints [-139.916, 60.325, -67.472, 139.696, 84.538, 4.616]
  Call Extruder(790.32530)
  MoveL 3105 to (-33.45, 162.37, 50.44) mm, rotated rx -180 ry 0 rz -180 deg; joints [-139.991, 60.331, -67.464, 139.771, 84.543, 4.599]
  MoveL 3106 to (-33.45, 162.37, 50.44) mm, rotated rx -180 ry 0 rz -180 deg; joints [-139.991, 60.331, -67.464, 139.771, 84.543, 4.599]
  Call Extruder(790.53263)
  MoveL 3107 to (-33.75, 162.2, 50.44) mm, rotated rx -180 ry 0 rz 180 deg; joints [-140.065, 60.338, -67.456, 139.847, 84.548, 4.583]
  MoveL 3108 to (-33.75, 162.2, 50.44) mm, rotated rx -180 ry 0 rz 180 deg; joints [-140.065, 60.338, -67.456, 139.847, 84.548, 4.583]
  Call Extruder(790.74074)
  MoveL 3109 to (-34.05, 162.02, 50.44) mm, rotated rx -180 ry 0 rz 180 deg; joints [-140.14, 60.344, -67.447, 139.923, 84.553, 4.566]
  MoveL 3110 to (-34.05, 162.02, 50.44) mm, rotated rx -180 ry 0 rz 180 deg; joints [-140.14, 60.344, -67.447, 139.923, 84.553, 4.566]
  Call Extruder(790.85846)
  MoveL 3111 to (-34.23, 161.92, 50.44) mm, rotated rx 180 ry 0 rz -180 deg; joints [-140.182, 60.348, -67.443, 139.966, 84.556, 4.557]
  MoveL 3112 to (-34.23, 161.92, 50.44) mm, rotated rx 180 ry 0 rz -180 deg; joints [-140.182, 60.348, -67.443, 139.966, 84.556, 4.557]
  Call Extruder(791.19129)
  MoveL 3113 to (-34.68, 161.59, 50.44) mm, rotated rx -180 ry 0 rz -180 deg; joints [-140.305, 60.355, -67.433, 140.089, 84.559, 4.534]
  MoveL 3114 to (-34.68, 161.59, 50.44) mm, rotated rx -180 ry 0 rz -180 deg; joints [-140.305, 60.355, -67.433, 140.089, 84.559, 4.534]
  Call Extruder(791.52530)
  MoveL 3115 to (-35.13, 161.27, 50.44) mm, rotated rx -180 ry 0 rz 180 deg; joints [-140.427, 60.363, -67.424, 140.213, 84.563, 4.512]
  MoveL 3116 to (-35.13, 161.27, 50.44) mm, rotated rx -180 ry 0 rz 180 deg; joints [-140.427, 60.363, -67.424, 140.213, 84.563, 4.512]
  Call Extruder(791.69289)
  MoveL 3117 to (-35.35, 161.1, 50.44) mm, rotated rx 180 ry 0 rz 180 deg; joints [-140.489, 60.366, -67.419, 140.275, 84.564, 4.501]
  Call Extruder(792.52220)
  MoveL 3118 to (-36.39, 160.19, 50.44) mm, rotated rx 180 ry 0 rz -180 deg; joints [-140.797, 60.378, -67.404, 140.585, 84.561, 4.454]
  Call Extruder(793.04443)
  MoveL 3119 to (-36.97, 159.54, 50.44) mm, rotated rx -180 ry 0 rz 180 deg; joints [-140.993, 60.38, -67.401, 140.782, 84.55, 4.432]
  Set speed (130.0 mm/s)
  MoveL 3120 to (-38.97, 156.78, 50.44) mm, rotated rx -180 ry 0 rz -180 deg; joints [-141.763, 60.372, -67.412, 141.552, 84.476, 4.37]
  MoveL 3121 to (-38.97, 156.79, 59.84) mm, rotated rx 180 ry 0 rz -180 deg; joints [-141.763, 61.778, -69.453, 141.512, 83.978, 4.768]
  Call Extruder(791.04443)
  Set speed (40.0 mm/s)
  MoveL 3122 to (-38.97, 156.79, 59.84) mm, rotated rx 180 ry 0 rz -180 deg; joints [-141.763, 61.778, -69.453, 141.512, 83.978, 4.768]
  Call Extruder(0.00000)
  Set speed (130.0 mm/s)
  MoveL 3123 to (-31.64, 163.21, 59.84) mm, rotated rx -180 ry 0 rz -180 deg; joints [-139.581, 61.69, -69.562, 139.313, 84.014, 5.123]
  Call Extruder(2.00000)
  Set speed (40.0 mm/s)
  MoveL 3124 to (-31.64, 163.21, 59.84) mm, rotated rx -180 ry 0 rz -180 deg; joints [-139.581, 61.69, -69.562, 139.313, 84.014, 5.123]
  Set speed (30.0 mm/s)
  MoveL 3125 to (-31.64, 163.21, 59.84) mm, rotated rx -180 ry 0 rz -180 deg; joints [-139.581, 61.69, -69.562, 139.313, 84.014, 5.123]
  Call Extruder(2.18198)
  MoveL 3126 to (-31.93, 163.09, 59.84) mm, rotated rx -180 ry 0 rz 180 deg; joints [-139.645, 61.697, -69.553, 139.378, 84.022, 5.105]
  MoveL 3127 to (-31.93, 163.09, 59.84) mm, rotated rx -180 ry 0 rz 180 deg; joints [-139.645, 61.697, -69.553, 139.378, 84.022, 5.105]
  Call Extruder(2.36471)
  MoveL 3128 to (-32.22, 162.96, 59.84) mm, rotated rx -180 ry 0 rz 180 deg; joints [-139.709, 61.705, -69.543, 139.443, 84.03, 5.087]
  MoveL 3129 to (-32.22, 162.96, 59.84) mm, rotated rx -180 ry 0 rz 180 deg; joints [-139.709, 61.705, -69.543, 139.443, 84.03, 5.087]
  Call Extruder(2.53513)
  MoveL 3130 to (-32.49, 162.85, 59.84) mm, rotated rx -180 ry 0 rz 180 deg; joints [-139.768, 61.713, -69.534, 139.504, 84.037, 5.07]
  MoveL 3131 to (-32.49, 162.85, 59.84) mm, rotated rx -180 ry 0 rz 180 deg; joints [-139.768, 61.713, -69.534, 139.504, 84.037, 5.07]
  Call Extruder(2.69310)
  MoveL 3132 to (-32.74, 162.74, 59.84) mm, rotated rx 180 ry 0 rz 180 deg; joints [-139.823, 61.719, -69.526, 139.56, 84.043, 5.054]
  MoveL 3133 to (-32.74, 162.74, 59.84) mm, rotated rx 180 ry 0 rz 180 deg; joints [-139.823, 61.719, -69.526, 139.56, 84.043, 5.054]
  Call Extruder(2.85168)
  MoveL 3134 to (-32.99, 162.64, 59.84) mm, rotated rx 180 ry 0 rz 180 deg; joints [-139.878, 61.726, -69.517, 139.616, 84.05, 5.039]
  MoveL 3135 to (-32.99, 162.64, 59.84) mm, rotated rx 180 ry 0 rz 180 deg; joints [-139.878, 61.726, -69.517, 139.616, 84.05, 5.039]
  Call Extruder(3.05785)
  MoveL 3136 to (-33.29, 162.46, 59.84) mm, rotated rx -180 ry 0 rz 180 deg; joints [-139.953, 61.733, -69.509, 139.692, 84.055, 5.022]
  MoveL 3137 to (-33.29, 162.46, 59.84) mm, rotated rx -180 ry 0 rz 180 deg; joints [-139.953, 61.733, -69.509, 139.692, 84.055, 5.022]
  Call Extruder(3.26479)
  MoveL 3138 to (-33.6, 162.29, 59.84) mm, rotated rx -180 ry 0 rz 180 deg; joints [-140.028, 61.739, -69.501, 139.768, 84.059, 5.004]
  MoveL 3139 to (-33.6, 162.29, 59.84) mm, rotated rx -180 ry 0 rz 180 deg; joints [-140.028, 61.739, -69.501, 139.768, 84.059, 5.004]
  Call Extruder(3.47251)
  MoveL 3140 to (-33.9, 162.11, 59.84) mm, rotated rx -180 ry 0 rz -180 deg; joints [-140.103, 61.746, -69.493, 139.844, 84.064, 4.987]
  MoveL 3141 to (-33.9, 162.11, 59.84) mm, rotated rx -180 ry 0 rz -180 deg; joints [-140.103, 61.746, -69.493, 139.844, 84.064, 4.987]
  Call Extruder(3.68101)
  MoveL 3142 to (-34.21, 161.94, 59.84) mm, rotated rx -180 ry 0 rz -180 deg; joints [-140.178, 61.753, -69.485, 139.92, 84.069, 4.97]
  MoveL 3143 to (-34.21, 161.94, 59.84) mm, rotated rx -180 ry 0 rz -180 deg; joints [-140.178, 61.753, -69.485, 139.92, 84.069, 4.97]
  Call Extruder(3.86055)
  MoveL 3144 to (-34.45, 161.76, 59.84) mm, rotated rx -180 ry 0 rz 180 deg; joints [-140.244, 61.757, -69.48, 139.987, 84.07, 4.957]
  MoveL 3145 to (-34.45, 161.76, 59.84) mm, rotated rx -180 ry 0 rz 180 deg; joints [-140.244, 61.757, -69.48, 139.987, 84.07, 4.957]
  Call Extruder(4.19399)
  MoveL 3146 to (-34.9, 161.43, 59.84) mm, rotated rx -180 ry 0 rz -180 deg; joints [-140.366, 61.764, -69.47, 140.111, 84.073, 4.933]
  MoveL 3147 to (-34.9, 161.43, 59.84) mm, rotated rx -180 ry 0 rz -180 deg; joints [-140.366, 61.764, -69.47, 140.111, 84.073, 4.933]
  Call Extruder(4.52861)
  MoveL 3148 to (-35.35, 161.1, 59.84) mm, rotated rx 180 ry 0 rz 180 deg; joints [-140.489, 61.772, -69.461, 140.234, 84.075, 4.909]
  Call Extruder(5.35652)
  MoveL 3149 to (-36.39, 160.19, 59.84) mm, rotated rx -180 ry 0 rz -180 deg; joints [-140.797, 61.784, -69.446, 140.545, 84.07, 4.86]
  Call Extruder(6.18445)
  MoveL 3150 to (-37.3, 159.15, 59.84) mm, rotated rx -180 ry 0 rz 180 deg; joints [-141.109, 61.787, -69.442, 140.858, 84.049, 4.823]
  Call Extruder(6.35176)
  MoveL 3151 to (-37.47, 158.93, 59.84) mm, rotated rx -180 ry 0 rz 180 deg; joints [-141.172, 61.786, -69.443, 140.921, 84.042, 4.818]
  MoveL 3152 to (-37.47, 158.93, 59.84) mm, rotated rx -180 ry 0 rz 180 deg; joints [-141.172, 61.786, -69.443, 140.921, 84.042, 4.818]
  Call Extruder(6.68519)
  MoveL 3153 to (-37.8, 158.48, 59.84) mm, rotated rx 180 ry 0 rz 180 deg; joints [-141.298, 61.785, -69.445, 141.047, 84.029, 4.807]
  MoveL 3154 to (-37.8, 158.48, 59.84) mm, rotated rx 180 ry 0 rz 180 deg; joints [-141.298, 61.785, -69.445, 141.047, 84.029, 4.807]
  Call Extruder(7.01744)
  MoveL 3155 to (-38.12, 158.02, 59.84) mm, rotated rx 180 ry 0 rz 180 deg; joints [-141.424, 61.784, -69.446, 141.173, 84.016, 4.796]
  MoveL 3156 to (-38.12, 158.02, 59.84) mm, rotated rx 180 ry 0 rz 180 deg; joints [-141.424, 61.784, -69.446, 141.173, 84.016, 4.796]
  Call Extruder(7.13511)
  MoveL 3157 to (-38.22, 157.85, 59.84) mm, rotated rx -180 ry 0 rz 180 deg; joints [-141.468, 61.782, -69.448, 141.217, 84.01, 4.793]
  MoveL 3158 to (-38.22, 157.85, 59.84) mm, rotated rx -180 ry 0 rz 180 deg; joints [-141.468, 61.782, -69.448, 141.217, 84.01, 4.793]
  Call Extruder(7.34283)
  MoveL 3159 to (-38.4, 157.55, 59.84) mm, rotated rx -180 ry 0 rz 180 deg; joints [-141.547, 61.779, -69.452, 141.295, 83.998, 4.789]
  MoveL 3160 to (-38.4, 157.55, 59.84) mm, rotated rx -180 ry 0 rz 180 deg; joints [-141.547, 61.779, -69.452, 141.295, 83.998, 4.789]
  Call Extruder(7.54978)
  MoveL 3161 to (-38.57, 157.25, 59.84) mm, rotated rx 180 ry 0 rz 180 deg; joints [-141.625, 61.776, -69.455, 141.374, 83.987, 4.785]
  MoveL 3162 to (-38.57, 157.25, 59.84) mm, rotated rx 180 ry 0 rz 180 deg; joints [-141.625, 61.776, -69.455, 141.374, 83.987, 4.785]
  Call Extruder(7.75595)
  MoveL 3163 to (-38.75, 156.94, 59.84) mm, rotated rx -180 ry 0 rz 180 deg; joints [-141.704, 61.773, -69.459, 141.452, 83.975, 4.78]
  MoveL 3164 to (-38.75, 156.94, 59.84) mm, rotated rx -180 ry 0 rz 180 deg; joints [-141.704, 61.773, -69.459, 141.452, 83.975, 4.78]
  Call Extruder(7.93763)
  MoveL 3165 to (-38.89, 156.66, 59.84) mm, rotated rx -180 ry 0 rz 180 deg; joints [-141.773, 61.77, -69.463, 141.521, 83.964, 4.778]
  MoveL 3166 to (-38.89, 156.66, 59.84) mm, rotated rx -180 ry 0 rz 180 deg; joints [-141.773, 61.77, -69.463, 141.521, 83.964, 4.778]
  Call Extruder(8.09561)
  MoveL 3167 to (-39, 156.42, 59.84) mm, rotated rx 180 ry 0 rz -180 deg; joints [-141.832, 61.766, -69.468, 141.58, 83.952, 4.777]
  MoveL 3168 to (-39, 156.42, 59.84) mm, rotated rx 180 ry 0 rz -180 deg; joints [-141.832, 61.766, -69.468, 141.58, 83.952, 4.777]
  Call Extruder(8.25300)
  MoveL 3169 to (-39.11, 156.17, 59.84) mm, rotated rx -180 ry 0 rz 180 deg; joints [-141.891, 61.763, -69.472, 141.638, 83.941, 4.776]
  MoveL 3170 to (-39.11, 156.17, 59.84) mm, rotated rx -180 ry 0 rz 180 deg; joints [-141.891, 61.763, -69.472, 141.638, 83.941, 4.776]
  Call Extruder(8.43572)
  MoveL 3171 to (-39.23, 155.87, 59.84) mm, rotated rx -180 ry 0 rz 180 deg; joints [-141.96, 61.758, -69.478, 141.707, 83.927, 4.775]
  MoveL 3172 to (-39.23, 155.87, 59.84) mm, rotated rx -180 ry 0 rz 180 deg; joints [-141.96, 61.758, -69.478, 141.707, 83.927, 4.775]
  Call Extruder(8.61768)
  MoveL 3173 to (-39.35, 155.58, 59.84) mm, rotated rx -180 ry 0 rz 180 deg; joints [-142.029, 61.753, -69.484, 141.775, 83.913, 4.774]
  MoveL 3174 to (-39.35, 155.58, 59.84) mm, rotated rx -180 ry 0 rz 180 deg; joints [-142.029, 61.753, -69.484, 141.775, 83.913, 4.774]
  Call Extruder(8.76501)
  MoveL 3175 to (-39.44, 155.34, 59.84) mm, rotated rx -180 ry 0 rz 180 deg; joints [-142.085, 61.749, -69.489, 141.83, 83.901, 4.774]
  MoveL 3176 to (-39.44, 155.34, 59.84) mm, rotated rx -180 ry 0 rz 180 deg; joints [-142.085, 61.749, -69.489, 141.83, 83.901, 4.774]
  Call Extruder(8.87825)
  MoveL 3177 to (-39.5, 155.15, 59.84) mm, rotated rx 180 ry 0 rz 180 deg; joints [-142.127, 61.745, -69.494, 141.872, 83.891, 4.775]
  MoveL 3178 to (-39.5, 155.15, 59.84) mm, rotated rx 180 ry 0 rz 180 deg; joints [-142.127, 61.745, -69.494, 141.872, 83.891, 4.775]
  Call Extruder(8.99104)
  MoveL 3179 to (-39.56, 154.97, 59.84) mm, rotated rx 180 ry 0 rz 180 deg; joints [-142.169, 61.742, -69.498, 141.914, 83.881, 4.776]
  MoveL 3180 to (-39.56, 154.97, 59.84) mm, rotated rx 180 ry 0 rz 180 deg; joints [-142.169, 61.742, -69.498, 141.914, 83.881, 4.776]
  Call Extruder(9.10338)
  MoveL 3181 to (-39.62, 154.78, 59.84) mm, rotated rx -180 ry 0 rz 180 deg; joints [-142.212, 61.738, -69.503, 141.956, 83.871, 4.776]
  MoveL 3182 to (-39.62, 154.78, 59.84) mm, rotated rx -180 ry 0 rz 180 deg; joints [-142.212, 61.738, -69.503, 141.956, 83.871, 4.776]
  Call Extruder(9.21528)
  MoveL 3183 to (-39.68, 154.59, 59.84) mm, rotated rx -180 ry 0 rz -180 deg; joints [-142.254, 61.734, -69.507, 141.998, 83.861, 4.777]
  MoveL 3184 to (-39.68, 154.59, 59.84) mm, rotated rx -180 ry 0 rz -180 deg; joints [-142.254, 61.734, -69.507, 141.998, 83.861, 4.777]
  Call Extruder(9.33668)
  MoveL 3185 to (-39.75, 154.38, 59.84) mm, rotated rx -180 ry 0 rz -180 deg; joints [-142.3, 61.73, -69.512, 142.043, 83.85, 4.777]
  MoveL 3186 to (-39.75, 154.38, 59.84) mm, rotated rx -180 ry 0 rz -180 deg; joints [-142.3, 61.73, -69.512, 142.043, 83.85, 4.777]
  Call Extruder(9.46748)
  MoveL 3187 to (-39.81, 154.16, 59.84) mm, rotated rx -180 ry 0 rz 180 deg; joints [-142.35, 61.726, -69.518, 142.092, 83.837, 4.778]
  MoveL 3188 to (-39.81, 154.16, 59.84) mm, rotated rx -180 ry 0 rz 180 deg; joints [-142.35, 61.726, -69.518, 142.092, 83.837, 4.778]
  Call Extruder(9.59771)
  MoveL 3189 to (-39.88, 153.94, 59.84) mm, rotated rx 180 ry 0 rz 180 deg; joints [-142.399, 61.721, -69.524, 142.141, 83.825, 4.779]
  MoveL 3190 to (-39.88, 153.94, 59.84) mm, rotated rx 180 ry 0 rz 180 deg; joints [-142.399, 61.721, -69.524, 142.141, 83.825, 4.779]
  Call Extruder(9.72737)
  MoveL 3191 to (-39.95, 153.71, 59.84) mm, rotated rx 180 ry 0 rz 180 deg; joints [-142.449, 61.716, -69.529, 142.19, 83.813, 4.78]
  MoveL 3192 to (-39.95, 153.71, 59.84) mm, rotated rx 180 ry 0 rz 180 deg; joints [-142.449, 61.716, -69.529, 142.19, 83.813, 4.78]
  Call Extruder(9.85647)
  MoveL 3193 to (-40.02, 153.49, 59.84) mm, rotated rx -180 ry 0 rz -180 deg; joints [-142.498, 61.712, -69.535, 142.239, 83.801, 4.781]
  MoveL 3194 to (-40.02, 153.49, 59.84) mm, rotated rx -180 ry 0 rz -180 deg; joints [-142.498, 61.712, -69.535, 142.239, 83.801, 4.781]
  Call Extruder(9.97156)
  MoveL 3195 to (-40.06, 153.28, 59.84) mm, rotated rx -180 ry 0 rz 180 deg; joints [-142.541, 61.707, -69.541, 142.282, 83.789, 4.783]
  MoveL 3196 to (-40.06, 153.28, 59.84) mm, rotated rx -180 ry 0 rz 180 deg; joints [-142.541, 61.707, -69.541, 142.282, 83.789, 4.783]
  Call Extruder(10.08619)
  MoveL 3197 to (-40.11, 153.08, 59.84) mm, rotated rx -180 ry 0 rz 180 deg; joints [-142.584, 61.702, -69.547, 142.324, 83.777, 4.785]
  MoveL 3198 to (-40.11, 153.08, 59.84) mm, rotated rx -180 ry 0 rz 180 deg; joints [-142.584, 61.702, -69.547, 142.324, 83.777, 4.785]
  Call Extruder(10.20037)
  MoveL 3199 to (-40.15, 152.88, 59.84) mm, rotated rx 180 ry 0 rz 180 deg; joints [-142.627, 61.697, -69.553, 142.366, 83.764, 4.787]
  MoveL 3200 to (-40.15, 152.88, 59.84) mm, rotated rx 180 ry 0 rz 180 deg; joints [-142.627, 61.697, -69.553, 142.366, 83.764, 4.787]
  Call Extruder(10.31410)
  MoveL 3201 to (-40.2, 152.67, 59.84) mm, rotated rx 180 ry 0 rz 180 deg; joints [-142.671, 61.692, -69.559, 142.409, 83.752, 4.789]
  MoveL 3202 to (-40.2, 152.67, 59.84) mm, rotated rx 180 ry 0 rz 180 deg; joints [-142.671, 61.692, -69.559, 142.409, 83.752, 4.789]
  Call Extruder(10.43953)
  MoveL 3203 to (-40.24, 152.44, 59.84) mm, rotated rx -180 ry 0 rz 180 deg; joints [-142.718, 61.687, -69.566, 142.456, 83.738, 4.792]
  MoveL 3204 to (-40.24, 152.44, 59.84) mm, rotated rx -180 ry 0 rz 180 deg; joints [-142.718, 61.687, -69.566, 142.456, 83.738, 4.792]
  Call Extruder(10.57650)
  MoveL 3205 to (-40.29, 152.2, 59.84) mm, rotated rx 180 ry 0 rz -180 deg; joints [-142.77, 61.681, -69.573, 142.507, 83.723, 4.794]
  MoveL 3206 to (-40.29, 152.2, 59.84) mm, rotated rx 180 ry 0 rz -180 deg; joints [-142.77, 61.681, -69.573, 142.507, 83.723, 4.794]
  Call Extruder(10.71287)
  MoveL 3207 to (-40.34, 151.95, 59.84) mm, rotated rx -180 ry 0 rz 180 deg; joints [-142.822, 61.675, -69.581, 142.558, 83.708, 4.797]
  MoveL 3208 to (-40.34, 151.95, 59.84) mm, rotated rx -180 ry 0 rz 180 deg; joints [-142.822, 61.675, -69.581, 142.558, 83.708, 4.797]
  Call Extruder(10.84862)
  MoveL 3209 to (-40.39, 151.7, 59.84) mm, rotated rx -180 ry 0 rz -180 deg; joints [-142.874, 61.668, -69.588, 142.61, 83.693, 4.799]
  MoveL 3210 to (-40.39, 151.7, 59.84) mm, rotated rx -180 ry 0 rz -180 deg; joints [-142.874, 61.668, -69.588, 142.61, 83.693, 4.799]
  Call Extruder(10.98377)
  MoveL 3211 to (-40.44, 151.45, 59.84) mm, rotated rx 180 ry 0 rz 180 deg; joints [-142.926, 61.662, -69.596, 142.661, 83.678, 4.802]
  MoveL 3212 to (-40.44, 151.45, 59.84) mm, rotated rx 180 ry 0 rz 180 deg; joints [-142.926, 61.662, -69.596, 142.661, 83.678, 4.802]
  Call Extruder(11.11831)
  MoveL 3213 to (-40.49, 151.2, 59.84) mm, rotated rx -180 ry 0 rz 180 deg; joints [-142.978, 61.656, -69.603, 142.712, 83.663, 4.805]
  MoveL 3214 to (-40.49, 151.2, 59.84) mm, rotated rx -180 ry 0 rz 180 deg; joints [-142.978, 61.656, -69.603, 142.712, 83.663, 4.805]
  Call Extruder(11.25223)
  MoveL 3215 to (-40.54, 150.95, 59.84) mm, rotated rx 180 ry 0 rz 180 deg; joints [-143.031, 61.65, -69.61, 142.764, 83.647, 4.807]
  MoveL 3216 to (-40.54, 150.95, 59.84) mm, rotated rx 180 ry 0 rz 180 deg; joints [-143.031, 61.65, -69.61, 142.764, 83.647, 4.807]
  Call Extruder(11.40009)
  MoveL 3217 to (-40.59, 150.67, 59.84) mm, rotated rx 180 ry 0 rz 180 deg; joints [-143.088, 61.643, -69.619, 142.82, 83.63, 4.81]
  MoveL 3218 to (-40.59, 150.67, 59.84) mm, rotated rx 180 ry 0 rz 180 deg; joints [-143.088, 61.643, -69.619, 142.82, 83.63, 4.81]
  Call Extruder(11.56181)
  MoveL 3219 to (-40.64, 150.37, 59.84) mm, rotated rx -180 ry 0 rz 180 deg; joints [-143.15, 61.635, -69.629, 142.882, 83.611, 4.814]
  MoveL 3220 to (-40.64, 150.37, 59.84) mm, rotated rx -180 ry 0 rz 180 deg; joints [-143.15, 61.635, -69.629, 142.882, 83.611, 4.814]
  Call Extruder(11.72281)
  MoveL 3221 to (-40.69, 150.06, 59.84) mm, rotated rx -180 ry 0 rz -180 deg; joints [-143.213, 61.627, -69.638, 142.943, 83.591, 4.818]
  MoveL 3222 to (-40.69, 150.06, 59.84) mm, rotated rx -180 ry 0 rz -180 deg; joints [-143.213, 61.627, -69.638, 142.943, 83.591, 4.818]
  Call Extruder(11.88308)
  MoveL 3223 to (-40.74, 149.76, 59.84) mm, rotated rx 180 ry 0 rz 180 deg; joints [-143.276, 61.619, -69.648, 143.005, 83.572, 4.821]
  MoveL 3224 to (-40.74, 149.76, 59.84) mm, rotated rx 180 ry 0 rz 180 deg; joints [-143.276, 61.619, -69.648, 143.005, 83.572, 4.821]
  Call Extruder(12.04262)
  MoveL 3225 to (-40.78, 149.45, 59.84) mm, rotated rx -180 ry 0 rz -180 deg; joints [-143.338, 61.611, -69.658, 143.066, 83.553, 4.825]
  MoveL 3226 to (-40.78, 149.45, 59.84) mm, rotated rx -180 ry 0 rz -180 deg; joints [-143.338, 61.611, -69.658, 143.066, 83.553, 4.825]
  Call Extruder(12.20144)
  MoveL 3227 to (-40.83, 149.14, 59.84) mm, rotated rx -180 ry 0 rz 180 deg; joints [-143.401, 61.603, -69.667, 143.128, 83.533, 4.829]
  MoveL 3228 to (-40.83, 149.14, 59.84) mm, rotated rx -180 ry 0 rz 180 deg; joints [-143.401, 61.603, -69.667, 143.128, 83.533, 4.829]
  Call Extruder(12.38010)
  MoveL 3229 to (-40.88, 148.8, 59.84) mm, rotated rx -180 ry 0 rz 180 deg; joints [-143.471, 61.593, -69.679, 143.197, 83.511, 4.833]
  MoveL 3230 to (-40.88, 148.8, 59.84) mm, rotated rx -180 ry 0 rz 180 deg; joints [-143.471, 61.593, -69.679, 143.197, 83.511, 4.833]
  Call Extruder(12.57854)
  MoveL 3231 to (-40.92, 148.41, 59.84) mm, rotated rx 180 ry 0 rz 180 deg; joints [-143.549, 61.583, -69.691, 143.274, 83.485, 4.839]
  MoveL 3232 to (-40.92, 148.41, 59.84) mm, rotated rx 180 ry 0 rz 180 deg; joints [-143.549, 61.583, -69.691, 143.274, 83.485, 4.839]
  Call Extruder(12.77612)
  MoveL 3233 to (-40.97, 148.02, 59.84) mm, rotated rx 180 ry 0 rz -180 deg; joints [-143.627, 61.572, -69.704, 143.35, 83.46, 4.844]
  MoveL 3234 to (-40.97, 148.02, 59.84) mm, rotated rx 180 ry 0 rz -180 deg; joints [-143.627, 61.572, -69.704, 143.35, 83.46, 4.844]
  Call Extruder(12.97282)
  MoveL 3235 to (-41.02, 147.64, 59.84) mm, rotated rx -180 ry 0 rz -180 deg; joints [-143.705, 61.561, -69.717, 143.427, 83.434, 4.849]
  MoveL 3236 to (-41.02, 147.64, 59.84) mm, rotated rx -180 ry 0 rz -180 deg; joints [-143.705, 61.561, -69.717, 143.427, 83.434, 4.849]
  Call Extruder(13.16866)
  MoveL 3237 to (-41.06, 147.25, 59.84) mm, rotated rx -180 ry 0 rz 180 deg; joints [-143.783, 61.55, -69.73, 143.503, 83.409, 4.854]
  MoveL 3238 to (-41.06, 147.25, 59.84) mm, rotated rx -180 ry 0 rz 180 deg; joints [-143.783, 61.55, -69.73, 143.503, 83.409, 4.854]
  Call Extruder(13.46406)
  MoveL 3239 to (-41.11, 146.66, 59.84) mm, rotated rx -180 ry 0 rz -180 deg; joints [-143.899, 61.533, -69.751, 143.617, 83.368, 4.864]
  MoveL 3240 to (-41.11, 146.66, 59.84) mm, rotated rx -180 ry 0 rz -180 deg; joints [-143.899, 61.533, -69.751, 143.617, 83.368, 4.864]
  Call Extruder(13.75812)
  MoveL 3241 to (-41.16, 146.07, 59.84) mm, rotated rx 180 ry 0 rz 180 deg; joints [-144.015, 61.516, -69.771, 143.73, 83.328, 4.873]
  MoveL 3242 to (-41.16, 146.07, 59.84) mm, rotated rx 180 ry 0 rz 180 deg; joints [-144.015, 61.516, -69.771, 143.73, 83.328, 4.873]
  Call Extruder(14.05086)
  MoveL 3243 to (-41.2, 145.48, 59.84) mm, rotated rx -180 ry 0 rz -180 deg; joints [-144.131, 61.498, -69.792, 143.845, 83.288, 4.882]
  MoveL 3244 to (-41.2, 145.48, 59.84) mm, rotated rx -180 ry 0 rz -180 deg; joints [-144.131, 61.498, -69.792, 143.845, 83.288, 4.882]
  Call Extruder(14.62431)
  MoveL 3245 to (-41.25, 144.32, 59.84) mm, rotated rx -180 ry 0 rz 180 deg; joints [-144.355, 61.462, -69.834, 144.064, 83.205, 4.902]
  MoveL 3246 to (-41.25, 144.32, 59.84) mm, rotated rx -180 ry 0 rz 180 deg; joints [-144.355, 61.462, -69.834, 144.064, 83.205, 4.902]
  Call Extruder(15.33827)
  MoveL 3247 to (-41.29, 142.86, 59.84) mm, rotated rx -180 ry 0 rz 180 deg; joints [-144.635, 61.416, -69.887, 144.338, 83.1, 4.927]
  Call Extruder(57.40310)
  MoveL 3248 to (-41.29, 57.14, 59.84) mm, rotated rx -180 ry 0 rz 180 deg; joints [-164.153, 59.07, -72.078, 163.757, 77.494, 3.61]
  Call Extruder(57.83165)
  MoveL 3249 to (-41.27, 56.26, 59.84) mm, rotated rx 180 ry 0 rz 180 deg; joints [-164.382, 59.052, -72.091, 163.99, 77.451, 3.568]
  MoveL 3250 to (-41.27, 56.26, 59.84) mm, rotated rx 180 ry 0 rz 180 deg; joints [-164.382, 59.052, -72.091, 163.99, 77.451, 3.568]
  Call Extruder(58.11773)
  MoveL 3251 to (-41.25, 55.68, 59.84) mm, rotated rx 180 ry 0 rz 180 deg; joints [-164.534, 59.04, -72.1, 164.144, 77.421, 3.54]
  MoveL 3252 to (-41.25, 55.68, 59.84) mm, rotated rx 180 ry 0 rz 180 deg; joints [-164.534, 59.04, -72.1, 164.144, 77.421, 3.54]
  Call Extruder(58.69247)
  MoveL 3253 to (-41.2, 54.52, 59.84) mm, rotated rx 180 ry 0 rz 180 deg; joints [-164.838, 59.016, -72.118, 164.452, 77.362, 3.483]
  MoveL 3254 to (-41.2, 54.52, 59.84) mm, rotated rx 180 ry 0 rz 180 deg; joints [-164.838, 59.016, -72.118, 164.452, 77.362, 3.483]
  Call Extruder(58.98587)
  MoveL 3255 to (-41.15, 53.93, 59.84) mm, rotated rx -180 ry 0 rz 180 deg; joints [-164.992, 59.003, -72.128, 164.608, 77.33, 3.455]
  MoveL 3256 to (-41.15, 53.93, 59.84) mm, rotated rx -180 ry 0 rz 180 deg; joints [-164.992, 59.003, -72.128, 164.608, 77.33, 3.455]
  Call Extruder(59.28060)
  MoveL 3257 to (-41.11, 53.34, 59.84) mm, rotated rx 180 ry 0 rz 180 deg; joints [-165.145, 58.989, -72.138, 164.763, 77.298, 3.427]
  MoveL 3258 to (-41.11, 53.34, 59.84) mm, rotated rx 180 ry 0 rz 180 deg; joints [-165.145, 58.989, -72.138, 164.763, 77.298, 3.427]
  Call Extruder(59.57666)
  MoveL 3259 to (-41.06, 52.75, 59.84) mm, rotated rx -180 ry 0 rz 180 deg; joints [-165.299, 58.976, -72.148, 164.919, 77.267, 3.399]
  MoveL 3260 to (-41.06, 52.75, 59.84) mm, rotated rx -180 ry 0 rz 180 deg; joints [-165.299, 58.976, -72.148, 164.919, 77.267, 3.399]
  Call Extruder(59.77294)
  MoveL 3261 to (-41.02, 52.37, 59.84) mm, rotated rx 180 ry 0 rz -180 deg; joints [-165.399, 58.966, -72.155, 165.021, 77.245, 3.381]
  MoveL 3262 to (-41.02, 52.37, 59.84) mm, rotated rx 180 ry 0 rz -180 deg; joints [-165.399, 58.966, -72.155, 165.021, 77.245, 3.381]
  Call Extruder(59.97008)
  MoveL 3263 to (-40.97, 51.98, 59.84) mm, rotated rx 180 ry 0 rz 180 deg; joints [-165.499, 58.957, -72.162, 165.123, 77.222, 3.362]
  MoveL 3264 to (-40.97, 51.98, 59.84) mm, rotated rx 180 ry 0 rz 180 deg; joints [-165.499, 58.957, -72.162, 165.123, 77.222, 3.362]
  Call Extruder(60.16808)
  MoveL 3265 to (-40.93, 51.59, 59.84) mm, rotated rx -180 ry 0 rz 180 deg; joints [-165.6, 58.947, -72.169, 165.224, 77.2, 3.344]
  MoveL 3266 to (-40.93, 51.59, 59.84) mm, rotated rx -180 ry 0 rz 180 deg; joints [-165.6, 58.947, -72.169, 165.224, 77.2, 3.344]
  Call Extruder(60.36696)
  MoveL 3267 to (-40.88, 51.2, 59.84) mm, rotated rx -180 ry 0 rz 180 deg; joints [-165.7, 58.937, -72.176, 165.327, 77.178, 3.326]
  MoveL 3268 to (-40.88, 51.2, 59.84) mm, rotated rx -180 ry 0 rz 180 deg; joints [-165.7, 58.937, -72.176, 165.327, 77.178, 3.326]
  Call Extruder(60.54604)
  MoveL 3269 to (-40.83, 50.86, 59.84) mm, rotated rx -180 ry 0 rz -180 deg; joints [-165.79, 58.928, -72.183, 165.417, 77.158, 3.309]
  MoveL 3270 to (-40.83, 50.86, 59.84) mm, rotated rx -180 ry 0 rz -180 deg; joints [-165.79, 58.928, -72.183, 165.417, 77.158, 3.309]
  Call Extruder(60.70522)
  MoveL 3271 to (-40.78, 50.55, 59.84) mm, rotated rx -180 ry 0 rz 180 deg; joints [-165.869, 58.92, -72.189, 165.497, 77.139, 3.295]
  MoveL 3272 to (-40.78, 50.55, 59.84) mm, rotated rx -180 ry 0 rz 180 deg; joints [-165.869, 58.92, -72.189, 165.497, 77.139, 3.295]
  Call Extruder(60.86512)
  MoveL 3273 to (-40.74, 50.24, 59.84) mm, rotated rx -180 ry 0 rz 180 deg; joints [-165.948, 58.912, -72.195, 165.577, 77.121, 3.281]
  MoveL 3274 to (-40.74, 50.24, 59.84) mm, rotated rx -180 ry 0 rz 180 deg; joints [-165.948, 58.912, -72.195, 165.577, 77.121, 3.281]
  Call Extruder(61.02576)
  MoveL 3275 to (-40.69, 49.94, 59.84) mm, rotated rx -180 ry 0 rz -180 deg; joints [-166.026, 58.903, -72.201, 165.657, 77.103, 3.267]
  MoveL 3276 to (-40.69, 49.94, 59.84) mm, rotated rx -180 ry 0 rz -180 deg; joints [-166.026, 58.903, -72.201, 165.657, 77.103, 3.267]
  Call Extruder(61.18712)
  MoveL 3277 to (-40.64, 49.63, 59.84) mm, rotated rx -180 ry 0 rz -180 deg; joints [-166.105, 58.895, -72.207, 165.737, 77.084, 3.252]
  MoveL 3278 to (-40.64, 49.63, 59.84) mm, rotated rx -180 ry 0 rz -180 deg; joints [-166.105, 58.895, -72.207, 165.737, 77.084, 3.252]
  Call Extruder(61.34921)
  MoveL 3279 to (-40.59, 49.33, 59.84) mm, rotated rx 180 ry 0 rz 180 deg; joints [-166.184, 58.887, -72.213, 165.817, 77.066, 3.238]
  MoveL 3280 to (-40.59, 49.33, 59.84) mm, rotated rx 180 ry 0 rz 180 deg; joints [-166.184, 58.887, -72.213, 165.817, 77.066, 3.238]
  Call Extruder(61.49741)
  MoveL 3281 to (-40.54, 49.05, 59.84) mm, rotated rx 180 ry 0 rz 180 deg; joints [-166.256, 58.879, -72.219, 165.89, 77.049, 3.225]
  MoveL 3282 to (-40.54, 49.05, 59.84) mm, rotated rx 180 ry 0 rz 180 deg; joints [-166.256, 58.879, -72.219, 165.89, 77.049, 3.225]
  Call Extruder(61.63164)
  MoveL 3283 to (-40.49, 48.8, 59.84) mm, rotated rx 180 ry 0 rz 180 deg; joints [-166.32, 58.872, -72.224, 165.955, 77.033, 3.213]
  MoveL 3284 to (-40.49, 48.8, 59.84) mm, rotated rx 180 ry 0 rz 180 deg; joints [-166.32, 58.872, -72.224, 165.955, 77.033, 3.213]
  Call Extruder(61.76648)
  MoveL 3285 to (-40.44, 48.55, 59.84) mm, rotated rx 180 ry 0 rz 180 deg; joints [-166.384, 58.864, -72.23, 166.019, 77.017, 3.201]
  MoveL 3286 to (-40.44, 48.55, 59.84) mm, rotated rx 180 ry 0 rz 180 deg; joints [-166.384, 58.864, -72.23, 166.019, 77.017, 3.201]
  Call Extruder(61.90193)
  MoveL 3287 to (-40.39, 48.3, 59.84) mm, rotated rx -180 ry 0 rz -180 deg; joints [-166.448, 58.857, -72.235, 166.084, 77.001, 3.19]
  MoveL 3288 to (-40.39, 48.3, 59.84) mm, rotated rx -180 ry 0 rz -180 deg; joints [-166.448, 58.857, -72.235, 166.084, 77.001, 3.19]
  Call Extruder(62.03799)
  MoveL 3289 to (-40.34, 48.05, 59.84) mm, rotated rx 180 ry 0 rz 180 deg; joints [-166.512, 58.85, -72.24, 166.149, 76.985, 3.178]
  MoveL 3290 to (-40.34, 48.05, 59.84) mm, rotated rx 180 ry 0 rz 180 deg; joints [-166.512, 58.85, -72.24, 166.149, 76.985, 3.178]
  Call Extruder(62.17466)
  MoveL 3291 to (-40.29, 47.8, 59.84) mm, rotated rx -180 ry 0 rz 180 deg; joints [-166.576, 58.842, -72.246, 166.215, 76.969, 3.166]
  MoveL 3292 to (-40.29, 47.8, 59.84) mm, rotated rx -180 ry 0 rz 180 deg; joints [-166.576, 58.842, -72.246, 166.215, 76.969, 3.166]
  Call Extruder(62.31194)
  MoveL 3293 to (-40.24, 47.55, 59.84) mm, rotated rx 180 ry 0 rz 180 deg; joints [-166.641, 58.835, -72.251, 166.28, 76.954, 3.155]
  MoveL 3294 to (-40.24, 47.55, 59.84) mm, rotated rx 180 ry 0 rz 180 deg; joints [-166.641, 58.835, -72.251, 166.28, 76.954, 3.155]
  Call Extruder(62.43761)
  MoveL 3295 to (-40.2, 47.33, 59.84) mm, rotated rx -180 ry 0 rz 180 deg; joints [-166.699, 58.828, -72.256, 166.339, 76.939, 3.144]
  MoveL 3296 to (-40.2, 47.33, 59.84) mm, rotated rx -180 ry 0 rz 180 deg; joints [-166.699, 58.828, -72.256, 166.339, 76.939, 3.144]
  Call Extruder(62.55157)
  MoveL 3297 to (-40.15, 47.12, 59.84) mm, rotated rx -180 ry 0 rz 180 deg; joints [-166.751, 58.822, -72.26, 166.392, 76.926, 3.134]
  MoveL 3298 to (-40.15, 47.12, 59.84) mm, rotated rx -180 ry 0 rz 180 deg; joints [-166.751, 58.822, -72.26, 166.392, 76.926, 3.134]
  Call Extruder(62.66597)
  MoveL 3299 to (-40.11, 46.92, 59.84) mm, rotated rx 180 ry 0 rz -180 deg; joints [-166.804, 58.816, -72.265, 166.445, 76.913, 3.125]
  MoveL 3300 to (-40.11, 46.92, 59.84) mm, rotated rx 180 ry 0 rz -180 deg; joints [-166.804, 58.816, -72.265, 166.445, 76.913, 3.125]
  Call Extruder(62.78083)
  MoveL 3301 to (-40.06, 46.72, 59.84) mm, rotated rx -180 ry 0 rz -180 deg; joints [-166.857, 58.81, -72.269, 166.499, 76.899, 3.115]
  MoveL 3302 to (-40.06, 46.72, 59.84) mm, rotated rx -180 ry 0 rz -180 deg; joints [-166.857, 58.81, -72.269, 166.499, 76.899, 3.115]
  Call Extruder(62.89615)
  MoveL 3303 to (-40.02, 46.51, 59.84) mm, rotated rx -180 ry 0 rz -180 deg; joints [-166.909, 58.803, -72.274, 166.552, 76.886, 3.105]
  MoveL 3304 to (-40.02, 46.51, 59.84) mm, rotated rx -180 ry 0 rz -180 deg; joints [-166.909, 58.803, -72.274, 166.552, 76.886, 3.105]
  Call Extruder(63.02553)
  MoveL 3305 to (-39.95, 46.29, 59.84) mm, rotated rx -180 ry 0 rz -180 deg; joints [-166.966, 58.795, -72.279, 166.609, 76.87, 3.095]
  MoveL 3306 to (-39.95, 46.29, 59.84) mm, rotated rx -180 ry 0 rz -180 deg; joints [-166.966, 58.795, -72.279, 166.609, 76.87, 3.095]
  Call Extruder(63.15547)
  MoveL 3307 to (-39.88, 46.06, 59.84) mm, rotated rx 180 ry 0 rz -180 deg; joints [-167.022, 58.787, -72.285, 166.667, 76.853, 3.086]
  MoveL 3308 to (-39.88, 46.06, 59.84) mm, rotated rx 180 ry 0 rz -180 deg; joints [-167.022, 58.787, -72.285, 166.667, 76.853, 3.086]
  Call Extruder(63.28598)
  MoveL 3309 to (-39.82, 45.84, 59.84) mm, rotated rx -180 ry 0 rz 180 deg; joints [-167.079, 58.779, -72.291, 166.724, 76.837, 3.076]
  MoveL 3310 to (-39.82, 45.84, 59.84) mm, rotated rx -180 ry 0 rz 180 deg; joints [-167.079, 58.779, -72.291, 166.724, 76.837, 3.076]
  Call Extruder(63.41706)
  MoveL 3311 to (-39.75, 45.62, 59.84) mm, rotated rx -180 ry 0 rz 180 deg; joints [-167.136, 58.771, -72.297, 166.782, 76.82, 3.066]
  MoveL 3312 to (-39.75, 45.62, 59.84) mm, rotated rx -180 ry 0 rz 180 deg; joints [-167.136, 58.771, -72.297, 166.782, 76.82, 3.066]
  Call Extruder(63.53870)
  MoveL 3313 to (-39.68, 45.41, 59.84) mm, rotated rx 180 ry 0 rz 180 deg; joints [-167.188, 58.764, -72.302, 166.834, 76.805, 3.056]
  MoveL 3314 to (-39.68, 45.41, 59.84) mm, rotated rx 180 ry 0 rz 180 deg; joints [-167.188, 58.764, -72.302, 166.834, 76.805, 3.056]
  Call Extruder(63.65083)
  MoveL 3315 to (-39.62, 45.22, 59.84) mm, rotated rx 180 ry 0 rz 180 deg; joints [-167.235, 58.757, -72.307, 166.882, 76.791, 3.048]
  MoveL 3316 to (-39.62, 45.22, 59.84) mm, rotated rx 180 ry 0 rz 180 deg; joints [-167.235, 58.757, -72.307, 166.882, 76.791, 3.048]
  Call Extruder(63.76340)
  MoveL 3317 to (-39.56, 45.03, 59.84) mm, rotated rx 180 ry 0 rz 180 deg; joints [-167.283, 58.75, -72.312, 166.931, 76.777, 3.04]
  MoveL 3318 to (-39.56, 45.03, 59.84) mm, rotated rx 180 ry 0 rz 180 deg; joints [-167.283, 58.75, -72.312, 166.931, 76.777, 3.04]
  Call Extruder(63.87641)
  MoveL 3319 to (-39.5, 44.85, 59.84) mm, rotated rx -180 ry 0 rz -180 deg; joints [-167.331, 58.743, -72.317, 166.979, 76.762, 3.031]
  MoveL 3320 to (-39.5, 44.85, 59.84) mm, rotated rx -180 ry 0 rz -180 deg; joints [-167.331, 58.743, -72.317, 166.979, 76.762, 3.031]
  Call Extruder(63.98987)
  MoveL 3321 to (-39.44, 44.66, 59.84) mm, rotated rx -180 ry 0 rz -180 deg; joints [-167.379, 58.736, -72.322, 167.028, 76.748, 3.023]
  MoveL 3322 to (-39.44, 44.66, 59.84) mm, rotated rx -180 ry 0 rz -180 deg; joints [-167.379, 58.736, -72.322, 167.028, 76.748, 3.023]
  Call Extruder(64.13751)
  MoveL 3323 to (-39.35, 44.42, 59.84) mm, rotated rx -180 ry 0 rz 180 deg; joints [-167.439, 58.726, -72.329, 167.088, 76.729, 3.012]
  MoveL 3324 to (-39.35, 44.42, 59.84) mm, rotated rx -180 ry 0 rz 180 deg; joints [-167.439, 58.726, -72.329, 167.088, 76.729, 3.012]
  Call Extruder(64.31985)
  MoveL 3325 to (-39.23, 44.13, 59.84) mm, rotated rx -180 ry 0 rz -180 deg; joints [-167.512, 58.713, -72.338, 167.162, 76.704, 3]
  MoveL 3326 to (-39.23, 44.13, 59.84) mm, rotated rx -180 ry 0 rz -180 deg; joints [-167.512, 58.713, -72.338, 167.162, 76.704, 3]
  Call Extruder(64.50294)
  MoveL 3327 to (-39.11, 43.83, 59.84) mm, rotated rx -180 ry 0 rz -180 deg; joints [-167.584, 58.701, -72.346, 167.235, 76.679, 2.988]
  MoveL 3328 to (-39.11, 43.83, 59.84) mm, rotated rx -180 ry 0 rz -180 deg; joints [-167.584, 58.701, -72.346, 167.235, 76.679, 2.988]
  Call Extruder(64.66063)
  MoveL 3329 to (-39, 43.58, 59.84) mm, rotated rx 180 ry 0 rz 180 deg; joints [-167.646, 58.69, -72.354, 167.298, 76.658, 2.978]
  MoveL 3330 to (-39, 43.58, 59.84) mm, rotated rx 180 ry 0 rz 180 deg; joints [-167.646, 58.69, -72.354, 167.298, 76.658, 2.978]
  Call Extruder(64.81891)
  MoveL 3331 to (-38.89, 43.33, 59.84) mm, rotated rx 180 ry 0 rz -180 deg; joints [-167.708, 58.679, -72.362, 167.361, 76.636, 2.967]
  MoveL 3332 to (-38.89, 43.33, 59.84) mm, rotated rx 180 ry 0 rz -180 deg; joints [-167.708, 58.679, -72.362, 167.361, 76.636, 2.967]
  Call Extruder(65.00094)
  MoveL 3333 to (-38.75, 43.06, 59.84) mm, rotated rx -180 ry 0 rz 180 deg; joints [-167.776, 58.665, -72.372, 167.429, 76.61, 2.956]
  MoveL 3334 to (-38.75, 43.06, 59.84) mm, rotated rx -180 ry 0 rz 180 deg; joints [-167.776, 58.665, -72.372, 167.429, 76.61, 2.956]
  Call Extruder(65.20749)
  MoveL 3335 to (-38.57, 42.75, 59.84) mm, rotated rx 180 ry 0 rz 180 deg; joints [-167.849, 58.649, -72.383, 167.503, 76.579, 2.945]
  MoveL 3336 to (-38.57, 42.75, 59.84) mm, rotated rx 180 ry 0 rz 180 deg; joints [-167.849, 58.649, -72.383, 167.503, 76.579, 2.945]
  Call Extruder(65.41482)
  MoveL 3337 to (-38.4, 42.45, 59.84) mm, rotated rx 180 ry 0 rz 180 deg; joints [-167.923, 58.632, -72.394, 167.577, 76.548, 2.934]
  MoveL 3338 to (-38.4, 42.45, 59.84) mm, rotated rx 180 ry 0 rz 180 deg; joints [-167.923, 58.632, -72.394, 167.577, 76.548, 2.934]
  Call Extruder(65.62294)
  MoveL 3339 to (-38.22, 42.15, 59.84) mm, rotated rx -180 ry 0 rz 180 deg; joints [-167.997, 58.616, -72.406, 167.651, 76.517, 2.922]
  MoveL 3340 to (-38.22, 42.15, 59.84) mm, rotated rx -180 ry 0 rz 180 deg; joints [-167.997, 58.616, -72.406, 167.651, 76.517, 2.922]
  Call Extruder(65.74065)
  MoveL 3341 to (-38.12, 41.98, 59.84) mm, rotated rx -180 ry 0 rz -180 deg; joints [-168.038, 58.606, -72.412, 167.693, 76.5, 2.916]
  MoveL 3342 to (-38.12, 41.98, 59.84) mm, rotated rx -180 ry 0 rz -180 deg; joints [-168.038, 58.606, -72.412, 167.693, 76.5, 2.916]
  Call Extruder(66.07350)
  MoveL 3343 to (-37.8, 41.52, 59.84) mm, rotated rx 180 ry 0 rz -180 deg; joints [-168.144, 58.577, -72.432, 167.799, 76.446, 2.901]
  MoveL 3344 to (-37.8, 41.52, 59.84) mm, rotated rx 180 ry 0 rz -180 deg; joints [-168.144, 58.577, -72.432, 167.799, 76.446, 2.901]
  Call Extruder(66.40753)
  MoveL 3345 to (-37.47, 41.07, 59.84) mm, rotated rx -180 ry 0 rz 180 deg; joints [-168.25, 58.548, -72.452, 167.906, 76.393, 2.886]
  MoveL 3346 to (-37.47, 41.07, 59.84) mm, rotated rx -180 ry 0 rz 180 deg; joints [-168.25, 58.548, -72.452, 167.906, 76.393, 2.886]
  Call Extruder(66.57512)
  MoveL 3347 to (-37.3, 40.85, 59.84) mm, rotated rx -180 ry 0 rz 180 deg; joints [-168.304, 58.534, -72.462, 167.96, 76.367, 2.878]
  Call Extruder(67.40443)
  MoveL 3348 to (-36.39, 39.81, 59.84) mm, rotated rx 180 ry 0 rz 180 deg; joints [-168.541, 58.456, -72.515, 168.197, 76.227, 2.848]
